	CONST robtarget Target_4220:=[[214.1,79.9,-54.2],[-0.0760679807605466,0.65526150182537,0.742837140883982,-0.114188478630225],[0,0,0,1],[9E+09,9E+09,9E+09,9E+09,9E+09,9E+09]];
	CONST robtarget Target_4230:=[[214.1,84.6,-54.5],[-0.0747816180925732,0.654610534044765,0.743306705241576,-0.115706094290646],[0,0,0,1],[9E+09,9E+09,9E+09,9E+09,9E+09,9E+09]];
	CONST robtarget Target_4240:=[[214.1,89.3,-54.9],[-0.073531882239943,0.653955613371436,0.743775907688082,-0.117185823276578],[0,0,0,1],[9E+09,9E+09,9E+09,9E+09,9E+09,9E+09]];
	CONST robtarget Target_4250:=[[214.1,94,-55.2],[-0.0722505034042859,0.653283696519975,0.744251094825556,-0.118703767716048],[0,0,0,1],[9E+09,9E+09,9E+09,9E+09,9E+09,9E+09]];
	CONST robtarget Target_4260:=[[214.1,98.7,-55.6],[-0.0709718230450671,0.652600969502751,0.744729273860509,-0.120221809971935],[0,0,0,1],[9E+09,9E+09,9E+09,9E+09,9E+09,9E+09]];
	CONST robtarget Target_4270:=[[214.1,103.4,-56.1],[-0.0697368456344226,0.651911675562493,0.745207121516542,-0.121713950175375],[0,0,0,1],[9E+09,9E+09,9E+09,9E+09,9E+09,9E+09]];
	CONST robtarget Target_4280:=[[214.1,108.1,-56.5],[-0.0684638092553564,0.65120670448846,0.745691861757032,-0.123232228580258],[0,0,0,1],[9E+09,9E+09,9E+09,9E+09,9E+09,9E+09]];
	CONST robtarget Target_4290:=[[214.1,112.9,-56.9],[-0.0672019671558274,0.650478513802981,0.746187667457493,-0.12476202797886],[0,0,0,1],[9E+09,9E+09,9E+09,9E+09,9E+09,9E+09]];
	CONST robtarget Target_4300:=[[214.1,117.6,-57.4],[-0.0659415982702471,0.649747743117887,0.746679097173527,-0.126292920525678],[0,0,0,1],[9E+09,9E+09,9E+09,9E+09,9E+09,9E+09]];
	CONST robtarget Target_4310:=[[214.1,122.3,-57.9],[-0.064724629163582,0.649009411435852,0.747171328797483,-0.127798715448665],[0,0,0,1],[9E+09,9E+09,9E+09,9E+09,9E+09,9E+09]];
	CONST robtarget Target_4320:=[[214.1,126.9,-58.4],[-0.0634688183068436,0.648264268897657,0.747662116568994,-0.129330994819074],[0,0,0,1],[9E+09,9E+09,9E+09,9E+09,9E+09,9E+09]];
	CONST robtarget Target_4330:=[[214.1,131.6,-59],[-0.0622181375236594,0.647496731507395,0.748165675952307,-0.13086255146968],[0,0,0,1],[9E+09,9E+09,9E+09,9E+09,9E+09,9E+09]];
	CONST robtarget Target_4340:=[[214.1,136.3,-59.5],[-0.0610108478057296,0.646720866963663,0.748670915845893,-0.132369393933289],[0,0,0,1],[9E+09,9E+09,9E+09,9E+09,9E+09,9E+09]];
	CONST robtarget Target_4350:=[[214.1,141,-60.1],[-0.0597731615365629,0.645924637221304,0.749183165378491,-0.133914588092245],[0,0,0,1],[9E+09,9E+09,9E+09,9E+09,9E+09,9E+09]];
	CONST robtarget Target_4360:=[[214.1,145.7,-60.7],[-0.0585391714057714,0.64511482893062,0.749700327915236,-0.135460109363351],[0,0,0,1],[9E+09,9E+09,9E+09,9E+09,9E+09,9E+09]];
	CONST robtarget Target_4370:=[[214.1,150.4,-61.3],[-0.0573428290888,0.644298492896021,0.750220650493769,-0.136967980114748],[0,0,0,1],[9E+09,9E+09,9E+09,9E+09,9E+09,9E+09]];
	CONST robtarget Target_4380:=[[214.1,155.2,-61.9],[-0.0561242209793799,0.643446414332673,0.750757651605653,-0.138527009126195],[0,0,0,1],[9E+09,9E+09,9E+09,9E+09,9E+09,9E+09]];
	CONST robtarget Target_4390:=[[214.1,159.9,-62.6],[-0.0549022874737579,0.642593676162974,0.751291241769304,-0.140073467245733],[0,0,0,1],[9E+09,9E+09,9E+09,9E+09,9E+09,9E+09]];
	CONST robtarget Target_4400:=[[214.1,164.6,-63.3],[-0.0536899475070816,0.641723004287069,0.751830248201575,-0.141634223246443],[0,0,0,1],[9E+09,9E+09,9E+09,9E+09,9E+09,9E+09]];
	CONST robtarget Target_4410:=[[214.1,169.3,-64],[-0.0525156005654393,0.640844533278809,0.752373783438205,-0.143157556066027],[0,0,0,1],[9E+09,9E+09,9E+09,9E+09,9E+09,9E+09]];
	CONST robtarget Target_4420:=[[214.1,174,-64.7],[-0.0513121794704837,0.639942656609551,0.752925495500269,-0.144719227178605],[0,0,0,1],[9E+09,9E+09,9E+09,9E+09,9E+09,9E+09]];
	CONST robtarget Target_4430:=[[214.1,178.7,-65.4],[-0.0501135494154515,0.639024535867129,0.753483945328914,-0.146281300432967],[0,0,0,1],[9E+09,9E+09,9E+09,9E+09,9E+09,9E+09]];
	CONST robtarget Target_4440:=[[214.1,183.4,-66.2],[-0.0489533985393246,0.638097583939901,0.754048044913025,-0.147805900099946],[0,0,0,1],[9E+09,9E+09,9E+09,9E+09,9E+09,9E+09]];
	CONST robtarget Target_4450:=[[214.1,188.1,-66.9],[-0.0477695461555189,0.63714240176872,0.754620547485047,-0.149383598972081],[0,0,0,1],[9E+09,9E+09,9E+09,9E+09,9E+09,9E+09]];
	CONST robtarget Target_4460:=[[214.1,192.8,-67.7],[-0.0465864465741739,0.636172890269665,0.755201164633342,-0.15094687018278],[0,0,0,1],[9E+09,9E+09,9E+09,9E+09,9E+09,9E+09]];
	CONST robtarget Target_4470:=[[214.1,197.5,-68.6],[-0.0454467284791908,0.635189863884349,0.755788257500963,-0.152487840540739],[0,0,0,1],[9E+09,9E+09,9E+09,9E+09,9E+09,9E+09]];
	CONST robtarget Target_4480:=[[214.1,202.2,-69.4],[-0.0442793548151249,0.634180120150372,0.756384963217846,-0.154067197550788],[0,0,0,1],[9E+09,9E+09,9E+09,9E+09,9E+09,9E+09]];
	CONST robtarget Target_4490:=[[214.1,206.9,-70.2],[-0.0431220973517324,0.633147478237495,0.756990026801105,-0.155662631498866],[0,0,0,1],[9E+09,9E+09,9E+09,9E+09,9E+09,9E+09]];
	CONST robtarget Target_4500:=[[214.1,211.6,-71.1],[-0.0419668302732848,0.632098525050186,0.757604653725667,-0.15724321428731],[0,0,0,1],[9E+09,9E+09,9E+09,9E+09,9E+09,9E+09]];
	CONST robtarget Target_4510:=[[214.1,216.3,-72],[-0.0408551063250609,0.631033669006859,0.758227646379614,-0.158802409089222],[0,0,0,1],[9E+09,9E+09,9E+09,9E+09,9E+09,9E+09]];
	CONST robtarget Target_4520:=[[214.1,221,-72.9],[-0.0397129990436774,0.629943181324887,0.758861906903818,-0.160384139675776],[0,0,0,1],[9E+09,9E+09,9E+09,9E+09,9E+09,9E+09]];
	CONST robtarget Target_4530:=[[214.1,225.7,-73.9],[-0.0385817057921211,0.628827052341548,0.759506197346856,-0.161982487983516],[0,0,0,1],[9E+09,9E+09,9E+09,9E+09,9E+09,9E+09]];
	CONST robtarget Target_4540:=[[214.1,230.4,-74.8],[-0.0374905350461494,0.627696847333574,0.760160850569989,-0.163543905084095],[0,0,0,1],[9E+09,9E+09,9E+09,9E+09,9E+09,9E+09]];
	CONST robtarget Target_4550:=[[214.1,235.1,-75.8],[-0.036377410933379,0.626530843722664,0.760827103763876,-0.165160237394547],[0,0,0,1],[9E+09,9E+09,9E+09,9E+09,9E+09,9E+09]];
	CONST robtarget Target_4560:=[[214.1,239.8,-76.8],[-0.0352685565372593,0.625344750184507,0.761505650251853,-0.166760957573877],[0,0,0,1],[9E+09,9E+09,9E+09,9E+09,9E+09,9E+09]];
	CONST robtarget Target_4570:=[[214.1,244.5,-77.8],[-0.0341712180146319,0.624129563242526,0.762196213319151,-0.168379180862828],[0,0,0,1],[9E+09,9E+09,9E+09,9E+09,9E+09,9E+09]];
	CONST robtarget Target_4580:=[[218.8,244.2,-79.1],[-0.0352789013652378,0.61925527973127,0.766168461703898,-0.168119558450798],[0,0,0,1],[9E+09,9E+09,9E+09,9E+09,9E+09,9E+09]];
	CONST robtarget Target_4590:=[[223.5,243.9,-80.3],[-0.0363420920703788,0.614382529573869,0.770085191873047,-0.167875420941287],[0,0,0,1],[9E+09,9E+09,9E+09,9E+09,9E+09,9E+09]];
	CONST robtarget Target_4600:=[[228.2,243.6,-81.6],[-0.0374001271246908,0.609513532222938,0.773944668193309,-0.167642879667832],[0,0,0,1],[9E+09,9E+09,9E+09,9E+09,9E+09,9E+09]];
	CONST robtarget Target_4610:=[[232.9,243.3,-82.8],[-0.0384493332726948,0.604654398226158,0.777746844476721,-0.167405356494801],[0,0,0,1],[9E+09,9E+09,9E+09,9E+09,9E+09,9E+09]];
	CONST robtarget Target_4620:=[[237.6,243,-84.1],[-0.0394894517675504,0.599806981726168,0.781491317968587,-0.167163057555683],[0,0,0,1],[9E+09,9E+09,9E+09,9E+09,9E+09,9E+09]];
	CONST robtarget Target_4630:=[[242.4,242.7,-85.3],[-0.0405424217596268,0.594868736122905,0.78525682561266,-0.166910804473919],[0,0,0,1],[9E+09,9E+09,9E+09,9E+09,9E+09,9E+09]];
	CONST robtarget Target_4640:=[[247.1,242.4,-86.6],[-0.0415634621821783,0.590050377687373,0.788883798273689,-0.166659482849602],[0,0,0,1],[9E+09,9E+09,9E+09,9E+09,9E+09,9E+09]];
	CONST robtarget Target_4650:=[[251.8,242.1,-87.8],[-0.0426055282136537,0.585257721214646,0.792452473450789,-0.166364798097438],[0,0,0,1],[9E+09,9E+09,9E+09,9E+09,9E+09,9E+09]];
	CONST robtarget Target_4660:=[[256.5,241.9,-89.1],[-0.0436128251589251,0.580445150786425,0.795984264824474,-0.166103577812228],[0,0,0,1],[9E+09,9E+09,9E+09,9E+09,9E+09,9E+09]];
	CONST robtarget Target_4670:=[[261.2,241.6,-90.3],[-0.044603962147879,0.575681451164459,0.799436294963406,-0.165840174991093],[0,0,0,1],[9E+09,9E+09,9E+09,9E+09,9E+09,9E+09]];
	CONST robtarget Target_4680:=[[265.9,241.2,-91.6],[-0.0455781193684878,0.570971841278474,0.802806750959846,-0.165575095093428],[0,0,0,1],[9E+09,9E+09,9E+09,9E+09,9E+09,9E+09]];
	CONST robtarget Target_4690:=[[270.7,241,-92.8],[-0.04657611167879,0.566118569710976,0.806236496288795,-0.165297135187669],[0,0,0,1],[9E+09,9E+09,9E+09,9E+09,9E+09,9E+09]];
	CONST robtarget Target_4700:=[[275.4,240.7,-94.1],[-0.0475652784406573,0.561433672938044,0.809512308110473,-0.164983630084364],[0,0,0,1],[9E+09,9E+09,9E+09,9E+09,9E+09,9E+09]];
	CONST robtarget Target_4710:=[[280.1,240.4,-95.3],[-0.0485138773113708,0.556766097158342,0.812729634716316,-0.164707187509133],[0,0,0,1],[9E+09,9E+09,9E+09,9E+09,9E+09,9E+09]];
	CONST robtarget Target_4720:=[[284.8,240.1,-96.6],[-0.0494516568369335,0.552125800136082,0.815889114350191,-0.164428061914728],[0,0,0,1],[9E+09,9E+09,9E+09,9E+09,9E+09,9E+09]];
	CONST robtarget Target_4730:=[[289.5,239.8,-97.8],[-0.0503785277368699,0.547513991237142,0.818991071679431,-0.164146452450295],[0,0,0,1],[9E+09,9E+09,9E+09,9E+09,9E+09,9E+09]];
	CONST robtarget Target_4740:=[[294.2,239.5,-99.1],[-0.0512944143707967,0.54293181630632,0.822035880563232,-0.163862555098194],[0,0,0,1],[9E+09,9E+09,9E+09,9E+09,9E+09,9E+09]];
	CONST robtarget Target_4750:=[[299,239.2,-100.3],[-0.0522188939240138,0.538281296648858,0.82508859631501,-0.163570293838167],[0,0,0,1],[9E+09,9E+09,9E+09,9E+09,9E+09,9E+09]];
	CONST robtarget Target_4760:=[[303.7,238.9,-101.6],[-0.0531406589164049,0.533770858467849,0.828019948764244,-0.16324124928732],[0,0,0,1],[9E+09,9E+09,9E+09,9E+09,9E+09,9E+09]];
    !***********************************************************
    !
    ! Module:  test
    !
    ! Description:
    !   <Insert description>
    !
    ! Author: ModuleWriter
    ! Version: 1.0
    !
    !***********************************************************


    !***********************************************************
    !
    ! Procedure main
    !
    !   This is the entry point of your program
    !
    !***********************************************************
    PROC main()
        Path_10;
      !Add your code here
    ENDPROC
      PROC Path_10()
SetDO drillDone,0;
MoveAbsJ jHome, v100, fine, tool0\WObj:= wobj0;
WaitTime 2;
confL \Off;
confJ \Off;
        MoveJ RelTool(Target_10,0,0,-10),v60,z10,DrillTool\WObj:=FakeWing;
SetDO drillDone,1;
WaitUntil drillDone = 0;
        MoveL Target_10,v30,fine,DrillTool\WObj:=FakeWing;
SetDO drillDone,1;
WaitUntil drillDone = 0;
        MoveL RelTool(Target_10,0,0,-10),v30,z10,DrillTool\WObj:=FakeWing;
        MoveL RelTool(Target_20,0,0,-10),v30,z10,DrillTool\WObj:=FakeWing;
        MoveL Target_20,v30,fine,DrillTool\WObj:=FakeWing;
SetDO drillDone,1;
WaitUntil drillDone = 0;
        MoveL RelTool(Target_20,0,0,-10),v30,z10,DrillTool\WObj:=FakeWing;
        MoveL RelTool(Target_30,0,0,-10),v30,z10,DrillTool\WObj:=FakeWing;
        MoveL Target_30,v30,fine,DrillTool\WObj:=FakeWing;
SetDO drillDone,1;
WaitUntil drillDone = 0;
        MoveL RelTool(Target_30,0,0,-10),v30,z10,DrillTool\WObj:=FakeWing;
        MoveL RelTool(Target_40,0,0,-10),v30,z10,DrillTool\WObj:=FakeWing;
        MoveL Target_40,v30,fine,DrillTool\WObj:=FakeWing;
SetDO drillDone,1;
WaitUntil drillDone = 0;
        MoveL RelTool(Target_40,0,0,-10),v30,z10,DrillTool\WObj:=FakeWing;
        MoveL RelTool(Target_50,0,0,-10),v30,z10,DrillTool\WObj:=FakeWing;
        MoveL Target_50,v30,fine,DrillTool\WObj:=FakeWing;
SetDO drillDone,1;
WaitUntil drillDone = 0;
        MoveL RelTool(Target_50,0,0,-10),v30,z10,DrillTool\WObj:=FakeWing;
        MoveL RelTool(Target_60,0,0,-10),v30,z10,DrillTool\WObj:=FakeWing;
        MoveL Target_60,v30,fine,DrillTool\WObj:=FakeWing;
SetDO drillDone,1;
WaitUntil drillDone = 0;
        MoveL RelTool(Target_60,0,0,-10),v30,z10,DrillTool\WObj:=FakeWing;
        MoveL RelTool(Target_70,0,0,-10),v30,z10,DrillTool\WObj:=FakeWing;
        MoveL Target_70,v30,fine,DrillTool\WObj:=FakeWing;
SetDO drillDone,1;
WaitUntil drillDone = 0;
        MoveL RelTool(Target_70,0,0,-10),v30,z10,DrillTool\WObj:=FakeWing;
        MoveL RelTool(Target_80,0,0,-10),v30,z10,DrillTool\WObj:=FakeWing;
        MoveL Target_80,v30,fine,DrillTool\WObj:=FakeWing;
SetDO drillDone,1;
WaitUntil drillDone = 0;
        MoveL RelTool(Target_80,0,0,-10),v30,z10,DrillTool\WObj:=FakeWing;
        MoveL RelTool(Target_90,0,0,-10),v30,z10,DrillTool\WObj:=FakeWing;
        MoveL Target_90,v30,fine,DrillTool\WObj:=FakeWing;
SetDO drillDone,1;
WaitUntil drillDone = 0;
        MoveL RelTool(Target_90,0,0,-10),v30,z10,DrillTool\WObj:=FakeWing;
        MoveL RelTool(Target_100,0,0,-10),v30,z10,DrillTool\WObj:=FakeWing;
        MoveL Target_100,v30,fine,DrillTool\WObj:=FakeWing;
SetDO drillDone,1;
WaitUntil drillDone = 0;
        MoveL RelTool(Target_100,0,0,-10),v30,z10,DrillTool\WObj:=FakeWing;
        MoveL RelTool(Target_110,0,0,-10),v30,z10,DrillTool\WObj:=FakeWing;
        MoveL Target_110,v30,fine,DrillTool\WObj:=FakeWing;
SetDO drillDone,1;
WaitUntil drillDone = 0;
        MoveL RelTool(Target_110,0,0,-10),v30,z10,DrillTool\WObj:=FakeWing;
        MoveL RelTool(Target_120,0,0,-10),v30,z10,DrillTool\WObj:=FakeWing;
        MoveL Target_120,v30,fine,DrillTool\WObj:=FakeWing;
SetDO drillDone,1;
WaitUntil drillDone = 0;
        MoveL RelTool(Target_120,0,0,-10),v30,z10,DrillTool\WObj:=FakeWing;
        MoveL RelTool(Target_130,0,0,-10),v30,z10,DrillTool\WObj:=FakeWing;
        MoveL Target_130,v30,fine,DrillTool\WObj:=FakeWing;
SetDO drillDone,1;
WaitUntil drillDone = 0;
        MoveL RelTool(Target_130,0,0,-10),v30,z10,DrillTool\WObj:=FakeWing;
        MoveL RelTool(Target_140,0,0,-10),v30,z10,DrillTool\WObj:=FakeWing;
        MoveL Target_140,v30,fine,DrillTool\WObj:=FakeWing;
SetDO drillDone,1;
WaitUntil drillDone = 0;
        MoveL RelTool(Target_140,0,0,-10),v30,z10,DrillTool\WObj:=FakeWing;
        MoveL RelTool(Target_150,0,0,-10),v30,z10,DrillTool\WObj:=FakeWing;
        MoveL Target_150,v30,fine,DrillTool\WObj:=FakeWing;
SetDO drillDone,1;
WaitUntil drillDone = 0;
        MoveL RelTool(Target_150,0,0,-10),v30,z10,DrillTool\WObj:=FakeWing;
        MoveL RelTool(Target_160,0,0,-10),v30,z10,DrillTool\WObj:=FakeWing;
        MoveL Target_160,v30,fine,DrillTool\WObj:=FakeWing;
SetDO drillDone,1;
WaitUntil drillDone = 0;
        MoveL RelTool(Target_160,0,0,-10),v30,z10,DrillTool\WObj:=FakeWing;
        MoveL RelTool(Target_170,0,0,-10),v30,z10,DrillTool\WObj:=FakeWing;
        MoveL Target_170,v30,fine,DrillTool\WObj:=FakeWing;
SetDO drillDone,1;
WaitUntil drillDone = 0;
        MoveL RelTool(Target_170,0,0,-10),v30,z10,DrillTool\WObj:=FakeWing;
        MoveL RelTool(Target_180,0,0,-10),v30,z10,DrillTool\WObj:=FakeWing;
        MoveL Target_180,v30,fine,DrillTool\WObj:=FakeWing;
SetDO drillDone,1;
WaitUntil drillDone = 0;
        MoveL RelTool(Target_180,0,0,-10),v30,z10,DrillTool\WObj:=FakeWing;
        MoveL RelTool(Target_190,0,0,-10),v30,z10,DrillTool\WObj:=FakeWing;
        MoveL Target_190,v30,fine,DrillTool\WObj:=FakeWing;
SetDO drillDone,1;
WaitUntil drillDone = 0;
        MoveL RelTool(Target_190,0,0,-10),v30,z10,DrillTool\WObj:=FakeWing;
        MoveL RelTool(Target_200,0,0,-10),v30,z10,DrillTool\WObj:=FakeWing;
        MoveL Target_200,v30,fine,DrillTool\WObj:=FakeWing;
SetDO drillDone,1;
WaitUntil drillDone = 0;
        MoveL RelTool(Target_200,0,0,-10),v30,z10,DrillTool\WObj:=FakeWing;
        MoveL RelTool(Target_210,0,0,-10),v30,z10,DrillTool\WObj:=FakeWing;
        MoveL Target_210,v30,fine,DrillTool\WObj:=FakeWing;
SetDO drillDone,1;
WaitUntil drillDone = 0;
        MoveL RelTool(Target_210,0,0,-10),v30,z10,DrillTool\WObj:=FakeWing;
        MoveL RelTool(Target_220,0,0,-10),v30,z10,DrillTool\WObj:=FakeWing;
        MoveL Target_220,v30,fine,DrillTool\WObj:=FakeWing;
SetDO drillDone,1;
WaitUntil drillDone = 0;
        MoveL RelTool(Target_220,0,0,-10),v30,z10,DrillTool\WObj:=FakeWing;
        MoveL RelTool(Target_230,0,0,-10),v30,z10,DrillTool\WObj:=FakeWing;
        MoveL Target_230,v30,fine,DrillTool\WObj:=FakeWing;
SetDO drillDone,1;
WaitUntil drillDone = 0;
        MoveL RelTool(Target_230,0,0,-10),v30,z10,DrillTool\WObj:=FakeWing;
        MoveL RelTool(Target_240,0,0,-10),v30,z10,DrillTool\WObj:=FakeWing;
        MoveL Target_240,v30,fine,DrillTool\WObj:=FakeWing;
SetDO drillDone,1;
WaitUntil drillDone = 0;
        MoveL RelTool(Target_240,0,0,-10),v30,z10,DrillTool\WObj:=FakeWing;
        MoveL RelTool(Target_250,0,0,-10),v30,z10,DrillTool\WObj:=FakeWing;
        MoveL Target_250,v30,fine,DrillTool\WObj:=FakeWing;
SetDO drillDone,1;
WaitUntil drillDone = 0;
        MoveL RelTool(Target_250,0,0,-10),v30,z10,DrillTool\WObj:=FakeWing;
        MoveL RelTool(Target_260,0,0,-10),v30,z10,DrillTool\WObj:=FakeWing;
        MoveL Target_260,v30,fine,DrillTool\WObj:=FakeWing;
SetDO drillDone,1;
WaitUntil drillDone = 0;
        MoveL RelTool(Target_260,0,0,-10),v30,z10,DrillTool\WObj:=FakeWing;
        MoveL RelTool(Target_270,0,0,-10),v30,z10,DrillTool\WObj:=FakeWing;
        MoveL Target_270,v30,fine,DrillTool\WObj:=FakeWing;
SetDO drillDone,1;
WaitUntil drillDone = 0;
        MoveL RelTool(Target_270,0,0,-10),v30,z10,DrillTool\WObj:=FakeWing;
        MoveL RelTool(Target_280,0,0,-10),v30,z10,DrillTool\WObj:=FakeWing;
        MoveL Target_280,v30,fine,DrillTool\WObj:=FakeWing;
SetDO drillDone,1;
WaitUntil drillDone = 0;
        MoveL RelTool(Target_280,0,0,-10),v30,z10,DrillTool\WObj:=FakeWing;
        MoveL RelTool(Target_290,0,0,-10),v30,z10,DrillTool\WObj:=FakeWing;
        MoveL Target_290,v30,fine,DrillTool\WObj:=FakeWing;
SetDO drillDone,1;
WaitUntil drillDone = 0;
        MoveL RelTool(Target_290,0,0,-10),v30,z10,DrillTool\WObj:=FakeWing;
        MoveL RelTool(Target_300,0,0,-10),v30,z10,DrillTool\WObj:=FakeWing;
        MoveL Target_300,v30,fine,DrillTool\WObj:=FakeWing;
SetDO drillDone,1;
WaitUntil drillDone = 0;
        MoveL RelTool(Target_300,0,0,-10),v30,z10,DrillTool\WObj:=FakeWing;
        MoveL RelTool(Target_310,0,0,-10),v30,z10,DrillTool\WObj:=FakeWing;
        MoveL Target_310,v30,fine,DrillTool\WObj:=FakeWing;
SetDO drillDone,1;
WaitUntil drillDone = 0;
        MoveL RelTool(Target_310,0,0,-10),v30,z10,DrillTool\WObj:=FakeWing;
        MoveL RelTool(Target_320,0,0,-10),v30,z10,DrillTool\WObj:=FakeWing;
        MoveL Target_320,v30,fine,DrillTool\WObj:=FakeWing;
SetDO drillDone,1;
WaitUntil drillDone = 0;
        MoveL RelTool(Target_320,0,0,-10),v30,z10,DrillTool\WObj:=FakeWing;
        MoveL RelTool(Target_330,0,0,-10),v30,z10,DrillTool\WObj:=FakeWing;
        MoveL Target_330,v30,fine,DrillTool\WObj:=FakeWing;
SetDO drillDone,1;
WaitUntil drillDone = 0;
        MoveL RelTool(Target_330,0,0,-10),v30,z10,DrillTool\WObj:=FakeWing;
        MoveL RelTool(Target_340,0,0,-10),v30,z10,DrillTool\WObj:=FakeWing;
        MoveL Target_340,v30,fine,DrillTool\WObj:=FakeWing;
SetDO drillDone,1;
WaitUntil drillDone = 0;
        MoveL RelTool(Target_340,0,0,-10),v30,z10,DrillTool\WObj:=FakeWing;
        MoveL RelTool(Target_350,0,0,-10),v30,z10,DrillTool\WObj:=FakeWing;
        MoveL Target_350,v30,fine,DrillTool\WObj:=FakeWing;
SetDO drillDone,1;
WaitUntil drillDone = 0;
        MoveL RelTool(Target_350,0,0,-10),v30,z10,DrillTool\WObj:=FakeWing;
        MoveL RelTool(Target_360,0,0,-10),v30,z10,DrillTool\WObj:=FakeWing;
        MoveL Target_360,v30,fine,DrillTool\WObj:=FakeWing;
SetDO drillDone,1;
WaitUntil drillDone = 0;
        MoveL RelTool(Target_360,0,0,-10),v30,z10,DrillTool\WObj:=FakeWing;
        MoveL RelTool(Target_370,0,0,-10),v30,z10,DrillTool\WObj:=FakeWing;
        MoveL Target_370,v30,fine,DrillTool\WObj:=FakeWing;
SetDO drillDone,1;
WaitUntil drillDone = 0;
        MoveL RelTool(Target_370,0,0,-10),v30,z10,DrillTool\WObj:=FakeWing;
        MoveL RelTool(Target_380,0,0,-10),v30,z10,DrillTool\WObj:=FakeWing;
        MoveL Target_380,v30,fine,DrillTool\WObj:=FakeWing;
SetDO drillDone,1;
WaitUntil drillDone = 0;
        MoveL RelTool(Target_380,0,0,-10),v30,z10,DrillTool\WObj:=FakeWing;
        MoveL RelTool(Target_390,0,0,-10),v30,z10,DrillTool\WObj:=FakeWing;
        MoveL Target_390,v30,fine,DrillTool\WObj:=FakeWing;
SetDO drillDone,1;
WaitUntil drillDone = 0;
        MoveL RelTool(Target_390,0,0,-10),v30,z10,DrillTool\WObj:=FakeWing;
        MoveL RelTool(Target_400,0,0,-10),v30,z10,DrillTool\WObj:=FakeWing;
        MoveL Target_400,v30,fine,DrillTool\WObj:=FakeWing;
SetDO drillDone,1;
WaitUntil drillDone = 0;
        MoveL RelTool(Target_400,0,0,-10),v30,z10,DrillTool\WObj:=FakeWing;
        MoveL RelTool(Target_410,0,0,-10),v30,z10,DrillTool\WObj:=FakeWing;
        MoveL Target_410,v30,fine,DrillTool\WObj:=FakeWing;
SetDO drillDone,1;
WaitUntil drillDone = 0;
        MoveL RelTool(Target_410,0,0,-10),v30,z10,DrillTool\WObj:=FakeWing;
        MoveL RelTool(Target_420,0,0,-10),v30,z10,DrillTool\WObj:=FakeWing;
        MoveL Target_420,v30,fine,DrillTool\WObj:=FakeWing;
SetDO drillDone,1;
WaitUntil drillDone = 0;
        MoveL RelTool(Target_420,0,0,-10),v30,z10,DrillTool\WObj:=FakeWing;
        MoveL RelTool(Target_430,0,0,-10),v30,z10,DrillTool\WObj:=FakeWing;
        MoveL Target_430,v30,fine,DrillTool\WObj:=FakeWing;
SetDO drillDone,1;
WaitUntil drillDone = 0;
        MoveL RelTool(Target_430,0,0,-10),v30,z10,DrillTool\WObj:=FakeWing;
        MoveL RelTool(Target_440,0,0,-10),v30,z10,DrillTool\WObj:=FakeWing;
        MoveL Target_440,v30,fine,DrillTool\WObj:=FakeWing;
SetDO drillDone,1;
WaitUntil drillDone = 0;
        MoveL RelTool(Target_440,0,0,-10),v30,z10,DrillTool\WObj:=FakeWing;
        MoveL RelTool(Target_450,0,0,-10),v30,z10,DrillTool\WObj:=FakeWing;
        MoveL Target_450,v30,fine,DrillTool\WObj:=FakeWing;
SetDO drillDone,1;
WaitUntil drillDone = 0;
        MoveL RelTool(Target_450,0,0,-10),v30,z10,DrillTool\WObj:=FakeWing;
        MoveL RelTool(Target_460,0,0,-10),v30,z10,DrillTool\WObj:=FakeWing;
        MoveL Target_460,v30,fine,DrillTool\WObj:=FakeWing;
SetDO drillDone,1;
WaitUntil drillDone = 0;
        MoveL RelTool(Target_460,0,0,-10),v30,z10,DrillTool\WObj:=FakeWing;
        MoveL RelTool(Target_470,0,0,-10),v30,z10,DrillTool\WObj:=FakeWing;
        MoveL Target_470,v30,fine,DrillTool\WObj:=FakeWing;
SetDO drillDone,1;
WaitUntil drillDone = 0;
        MoveL RelTool(Target_470,0,0,-10),v30,z10,DrillTool\WObj:=FakeWing;
        MoveL RelTool(Target_480,0,0,-10),v30,z10,DrillTool\WObj:=FakeWing;
        MoveL Target_480,v30,fine,DrillTool\WObj:=FakeWing;
SetDO drillDone,1;
WaitUntil drillDone = 0;
        MoveL RelTool(Target_480,0,0,-10),v30,z10,DrillTool\WObj:=FakeWing;
        MoveL RelTool(Target_490,0,0,-10),v30,z10,DrillTool\WObj:=FakeWing;
        MoveL Target_490,v30,fine,DrillTool\WObj:=FakeWing;
SetDO drillDone,1;
WaitUntil drillDone = 0;
        MoveL RelTool(Target_490,0,0,-10),v30,z10,DrillTool\WObj:=FakeWing;
        MoveL RelTool(Target_500,0,0,-10),v30,z10,DrillTool\WObj:=FakeWing;
        MoveL Target_500,v30,fine,DrillTool\WObj:=FakeWing;
SetDO drillDone,1;
WaitUntil drillDone = 0;
        MoveL RelTool(Target_500,0,0,-10),v30,z10,DrillTool\WObj:=FakeWing;
        MoveL RelTool(Target_510,0,0,-10),v30,z10,DrillTool\WObj:=FakeWing;
        MoveL Target_510,v30,fine,DrillTool\WObj:=FakeWing;
SetDO drillDone,1;
WaitUntil drillDone = 0;
        MoveL RelTool(Target_510,0,0,-10),v30,z10,DrillTool\WObj:=FakeWing;
        MoveL RelTool(Target_520,0,0,-10),v30,z10,DrillTool\WObj:=FakeWing;
        MoveL Target_520,v30,fine,DrillTool\WObj:=FakeWing;
SetDO drillDone,1;
WaitUntil drillDone = 0;
        MoveL RelTool(Target_520,0,0,-10),v30,z10,DrillTool\WObj:=FakeWing;
        MoveL RelTool(Target_530,0,0,-10),v30,z10,DrillTool\WObj:=FakeWing;
        MoveL Target_530,v30,fine,DrillTool\WObj:=FakeWing;
SetDO drillDone,1;
WaitUntil drillDone = 0;
        MoveL RelTool(Target_530,0,0,-10),v30,z10,DrillTool\WObj:=FakeWing;
        MoveL RelTool(Target_540,0,0,-10),v30,z10,DrillTool\WObj:=FakeWing;
        MoveL Target_540,v30,fine,DrillTool\WObj:=FakeWing;
SetDO drillDone,1;
WaitUntil drillDone = 0;
        MoveL RelTool(Target_540,0,0,-10),v30,z10,DrillTool\WObj:=FakeWing;
        MoveL RelTool(Target_550,0,0,-10),v30,z10,DrillTool\WObj:=FakeWing;
        MoveL Target_550,v30,fine,DrillTool\WObj:=FakeWing;
SetDO drillDone,1;
WaitUntil drillDone = 0;
        MoveL RelTool(Target_550,0,0,-10),v30,z10,DrillTool\WObj:=FakeWing;
        MoveL RelTool(Target_560,0,0,-10),v30,z10,DrillTool\WObj:=FakeWing;
        MoveL Target_560,v30,fine,DrillTool\WObj:=FakeWing;
SetDO drillDone,1;
WaitUntil drillDone = 0;
        MoveL RelTool(Target_560,0,0,-10),v30,z10,DrillTool\WObj:=FakeWing;
        MoveL RelTool(Target_570,0,0,-10),v30,z10,DrillTool\WObj:=FakeWing;
        MoveL Target_570,v30,fine,DrillTool\WObj:=FakeWing;
SetDO drillDone,1;
WaitUntil drillDone = 0;
        MoveL RelTool(Target_570,0,0,-10),v30,z10,DrillTool\WObj:=FakeWing;
        MoveL RelTool(Target_580,0,0,-10),v30,z10,DrillTool\WObj:=FakeWing;
        MoveL Target_580,v30,fine,DrillTool\WObj:=FakeWing;
SetDO drillDone,1;
WaitUntil drillDone = 0;
        MoveL RelTool(Target_580,0,0,-10),v30,z10,DrillTool\WObj:=FakeWing;
        MoveL RelTool(Target_590,0,0,-10),v30,z10,DrillTool\WObj:=FakeWing;
        MoveL Target_590,v30,fine,DrillTool\WObj:=FakeWing;
SetDO drillDone,1;
WaitUntil drillDone = 0;
        MoveL RelTool(Target_590,0,0,-10),v30,z10,DrillTool\WObj:=FakeWing;
        MoveL RelTool(Target_600,0,0,-10),v30,z10,DrillTool\WObj:=FakeWing;
        MoveL Target_600,v30,fine,DrillTool\WObj:=FakeWing;
SetDO drillDone,1;
WaitUntil drillDone = 0;
        MoveL RelTool(Target_600,0,0,-10),v30,z10,DrillTool\WObj:=FakeWing;
        MoveL RelTool(Target_610,0,0,-10),v30,z10,DrillTool\WObj:=FakeWing;
        MoveL Target_610,v30,fine,DrillTool\WObj:=FakeWing;
SetDO drillDone,1;
WaitUntil drillDone = 0;
        MoveL RelTool(Target_610,0,0,-10),v30,z10,DrillTool\WObj:=FakeWing;
        MoveL RelTool(Target_620,0,0,-10),v30,z10,DrillTool\WObj:=FakeWing;
        MoveL Target_620,v30,fine,DrillTool\WObj:=FakeWing;
SetDO drillDone,1;
WaitUntil drillDone = 0;
        MoveL RelTool(Target_620,0,0,-10),v30,z10,DrillTool\WObj:=FakeWing;
        MoveL RelTool(Target_630,0,0,-10),v30,z10,DrillTool\WObj:=FakeWing;
        MoveL Target_630,v30,fine,DrillTool\WObj:=FakeWing;
SetDO drillDone,1;
WaitUntil drillDone = 0;
        MoveL RelTool(Target_630,0,0,-10),v30,z10,DrillTool\WObj:=FakeWing;
        MoveL RelTool(Target_640,0,0,-10),v30,z10,DrillTool\WObj:=FakeWing;
        MoveL Target_640,v30,fine,DrillTool\WObj:=FakeWing;
SetDO drillDone,1;
WaitUntil drillDone = 0;
        MoveL RelTool(Target_640,0,0,-10),v30,z10,DrillTool\WObj:=FakeWing;
        MoveL RelTool(Target_650,0,0,-10),v30,z10,DrillTool\WObj:=FakeWing;
        MoveL Target_650,v30,fine,DrillTool\WObj:=FakeWing;
SetDO drillDone,1;
WaitUntil drillDone = 0;
        MoveL RelTool(Target_650,0,0,-10),v30,z10,DrillTool\WObj:=FakeWing;
        MoveL RelTool(Target_660,0,0,-10),v30,z10,DrillTool\WObj:=FakeWing;
        MoveL Target_660,v30,fine,DrillTool\WObj:=FakeWing;
SetDO drillDone,1;
WaitUntil drillDone = 0;
        MoveL RelTool(Target_660,0,0,-10),v30,z10,DrillTool\WObj:=FakeWing;
        MoveL RelTool(Target_670,0,0,-10),v30,z10,DrillTool\WObj:=FakeWing;
        MoveL Target_670,v30,fine,DrillTool\WObj:=FakeWing;
SetDO drillDone,1;
WaitUntil drillDone = 0;
        MoveL RelTool(Target_670,0,0,-10),v30,z10,DrillTool\WObj:=FakeWing;
        MoveL RelTool(Target_680,0,0,-10),v30,z10,DrillTool\WObj:=FakeWing;
        MoveL Target_680,v30,fine,DrillTool\WObj:=FakeWing;
SetDO drillDone,1;
WaitUntil drillDone = 0;
        MoveL RelTool(Target_680,0,0,-10),v30,z10,DrillTool\WObj:=FakeWing;
        MoveL RelTool(Target_690,0,0,-10),v30,z10,DrillTool\WObj:=FakeWing;
        MoveL Target_690,v30,fine,DrillTool\WObj:=FakeWing;
SetDO drillDone,1;
WaitUntil drillDone = 0;
        MoveL RelTool(Target_690,0,0,-10),v30,z10,DrillTool\WObj:=FakeWing;
        MoveL RelTool(Target_700,0,0,-10),v30,z10,DrillTool\WObj:=FakeWing;
        MoveL Target_700,v30,fine,DrillTool\WObj:=FakeWing;
SetDO drillDone,1;
WaitUntil drillDone = 0;
        MoveL RelTool(Target_700,0,0,-10),v30,z10,DrillTool\WObj:=FakeWing;
        MoveL RelTool(Target_710,0,0,-10),v30,z10,DrillTool\WObj:=FakeWing;
        MoveL Target_710,v30,fine,DrillTool\WObj:=FakeWing;
SetDO drillDone,1;
WaitUntil drillDone = 0;
        MoveL RelTool(Target_710,0,0,-10),v30,z10,DrillTool\WObj:=FakeWing;
        MoveL RelTool(Target_720,0,0,-10),v30,z10,DrillTool\WObj:=FakeWing;
        MoveL Target_720,v30,fine,DrillTool\WObj:=FakeWing;
SetDO drillDone,1;
WaitUntil drillDone = 0;
        MoveL RelTool(Target_720,0,0,-10),v30,z10,DrillTool\WObj:=FakeWing;
        MoveL RelTool(Target_730,0,0,-10),v30,z10,DrillTool\WObj:=FakeWing;
        MoveL Target_730,v30,fine,DrillTool\WObj:=FakeWing;
SetDO drillDone,1;
WaitUntil drillDone = 0;
        MoveL RelTool(Target_730,0,0,-10),v30,z10,DrillTool\WObj:=FakeWing;
        MoveL RelTool(Target_740,0,0,-10),v30,z10,DrillTool\WObj:=FakeWing;
        MoveL Target_740,v30,fine,DrillTool\WObj:=FakeWing;
SetDO drillDone,1;
WaitUntil drillDone = 0;
        MoveL RelTool(Target_740,0,0,-10),v30,z10,DrillTool\WObj:=FakeWing;
        MoveL RelTool(Target_750,0,0,-10),v30,z10,DrillTool\WObj:=FakeWing;
        MoveL Target_750,v30,fine,DrillTool\WObj:=FakeWing;
SetDO drillDone,1;
WaitUntil drillDone = 0;
        MoveL RelTool(Target_750,0,0,-10),v30,z10,DrillTool\WObj:=FakeWing;
        MoveL RelTool(Target_760,0,0,-10),v30,z10,DrillTool\WObj:=FakeWing;
        MoveL Target_760,v30,fine,DrillTool\WObj:=FakeWing;
SetDO drillDone,1;
WaitUntil drillDone = 0;
        MoveL RelTool(Target_760,0,0,-10),v30,z10,DrillTool\WObj:=FakeWing;
        MoveL RelTool(Target_770,0,0,-10),v30,z10,DrillTool\WObj:=FakeWing;
        MoveL Target_770,v30,fine,DrillTool\WObj:=FakeWing;
SetDO drillDone,1;
WaitUntil drillDone = 0;
        MoveL RelTool(Target_770,0,0,-10),v30,z10,DrillTool\WObj:=FakeWing;
        MoveL RelTool(Target_780,0,0,-10),v30,z10,DrillTool\WObj:=FakeWing;
        MoveL Target_780,v30,fine,DrillTool\WObj:=FakeWing;
SetDO drillDone,1;
WaitUntil drillDone = 0;
        MoveL RelTool(Target_780,0,0,-10),v30,z10,DrillTool\WObj:=FakeWing;
        MoveL RelTool(Target_790,0,0,-10),v30,z10,DrillTool\WObj:=FakeWing;
        MoveL Target_790,v30,fine,DrillTool\WObj:=FakeWing;
SetDO drillDone,1;
WaitUntil drillDone = 0;
        MoveL RelTool(Target_790,0,0,-10),v30,z10,DrillTool\WObj:=FakeWing;
        MoveL RelTool(Target_800,0,0,-10),v30,z10,DrillTool\WObj:=FakeWing;
        MoveL Target_800,v30,fine,DrillTool\WObj:=FakeWing;
SetDO drillDone,1;
WaitUntil drillDone = 0;
        MoveL RelTool(Target_800,0,0,-10),v30,z10,DrillTool\WObj:=FakeWing;
        MoveL RelTool(Target_810,0,0,-10),v30,z10,DrillTool\WObj:=FakeWing;
        MoveL Target_810,v30,fine,DrillTool\WObj:=FakeWing;
SetDO drillDone,1;
WaitUntil drillDone = 0;
        MoveL RelTool(Target_810,0,0,-10),v30,z10,DrillTool\WObj:=FakeWing;
        MoveL RelTool(Target_820,0,0,-10),v30,z10,DrillTool\WObj:=FakeWing;
        MoveL Target_820,v30,fine,DrillTool\WObj:=FakeWing;
SetDO drillDone,1;
WaitUntil drillDone = 0;
        MoveL RelTool(Target_820,0,0,-10),v30,z10,DrillTool\WObj:=FakeWing;
        MoveL RelTool(Target_830,0,0,-10),v30,z10,DrillTool\WObj:=FakeWing;
        MoveL Target_830,v30,fine,DrillTool\WObj:=FakeWing;
SetDO drillDone,1;
WaitUntil drillDone = 0;
        MoveL RelTool(Target_830,0,0,-10),v30,z10,DrillTool\WObj:=FakeWing;
        MoveL RelTool(Target_840,0,0,-10),v30,z10,DrillTool\WObj:=FakeWing;
        MoveL Target_840,v30,fine,DrillTool\WObj:=FakeWing;
SetDO drillDone,1;
WaitUntil drillDone = 0;
        MoveL RelTool(Target_840,0,0,-10),v30,z10,DrillTool\WObj:=FakeWing;
        MoveL RelTool(Target_850,0,0,-10),v30,z10,DrillTool\WObj:=FakeWing;
        MoveL Target_850,v30,fine,DrillTool\WObj:=FakeWing;
SetDO drillDone,1;
WaitUntil drillDone = 0;
        MoveL RelTool(Target_850,0,0,-10),v30,z10,DrillTool\WObj:=FakeWing;
        MoveL RelTool(Target_860,0,0,-10),v30,z10,DrillTool\WObj:=FakeWing;
        MoveL Target_860,v30,fine,DrillTool\WObj:=FakeWing;
SetDO drillDone,1;
WaitUntil drillDone = 0;
        MoveL RelTool(Target_860,0,0,-10),v30,z10,DrillTool\WObj:=FakeWing;
        MoveL RelTool(Target_870,0,0,-10),v30,z10,DrillTool\WObj:=FakeWing;
        MoveL Target_870,v30,fine,DrillTool\WObj:=FakeWing;
SetDO drillDone,1;
WaitUntil drillDone = 0;
        MoveL RelTool(Target_870,0,0,-10),v30,z10,DrillTool\WObj:=FakeWing;
        MoveL RelTool(Target_880,0,0,-10),v30,z10,DrillTool\WObj:=FakeWing;
        MoveL Target_880,v30,fine,DrillTool\WObj:=FakeWing;
SetDO drillDone,1;
WaitUntil drillDone = 0;
        MoveL RelTool(Target_880,0,0,-10),v30,z10,DrillTool\WObj:=FakeWing;
        MoveL RelTool(Target_890,0,0,-10),v30,z10,DrillTool\WObj:=FakeWing;
        MoveL Target_890,v30,fine,DrillTool\WObj:=FakeWing;
SetDO drillDone,1;
WaitUntil drillDone = 0;
        MoveL RelTool(Target_890,0,0,-10),v30,z10,DrillTool\WObj:=FakeWing;
        MoveL RelTool(Target_900,0,0,-10),v30,z10,DrillTool\WObj:=FakeWing;
        MoveL Target_900,v30,fine,DrillTool\WObj:=FakeWing;
SetDO drillDone,1;
WaitUntil drillDone = 0;
        MoveL RelTool(Target_900,0,0,-10),v30,z10,DrillTool\WObj:=FakeWing;
        MoveL RelTool(Target_910,0,0,-10),v30,z10,DrillTool\WObj:=FakeWing;
        MoveL Target_910,v30,fine,DrillTool\WObj:=FakeWing;
SetDO drillDone,1;
WaitUntil drillDone = 0;
        MoveL RelTool(Target_910,0,0,-10),v30,z10,DrillTool\WObj:=FakeWing;
        MoveL RelTool(Target_920,0,0,-10),v30,z10,DrillTool\WObj:=FakeWing;
        MoveL Target_920,v30,fine,DrillTool\WObj:=FakeWing;
SetDO drillDone,1;
WaitUntil drillDone = 0;
        MoveL RelTool(Target_920,0,0,-10),v30,z10,DrillTool\WObj:=FakeWing;
        MoveL RelTool(Target_930,0,0,-10),v30,z10,DrillTool\WObj:=FakeWing;
        MoveL Target_930,v30,fine,DrillTool\WObj:=FakeWing;
SetDO drillDone,1;
WaitUntil drillDone = 0;
        MoveL RelTool(Target_930,0,0,-10),v30,z10,DrillTool\WObj:=FakeWing;
        MoveL RelTool(Target_940,0,0,-10),v30,z10,DrillTool\WObj:=FakeWing;
        MoveL Target_940,v30,fine,DrillTool\WObj:=FakeWing;
SetDO drillDone,1;
WaitUntil drillDone = 0;
        MoveL RelTool(Target_940,0,0,-10),v30,z10,DrillTool\WObj:=FakeWing;
        MoveL RelTool(Target_950,0,0,-10),v30,z10,DrillTool\WObj:=FakeWing;
        MoveL Target_950,v30,fine,DrillTool\WObj:=FakeWing;
SetDO drillDone,1;
WaitUntil drillDone = 0;
        MoveL RelTool(Target_950,0,0,-10),v30,z10,DrillTool\WObj:=FakeWing;
        MoveL RelTool(Target_960,0,0,-10),v30,z10,DrillTool\WObj:=FakeWing;
        MoveL Target_960,v30,fine,DrillTool\WObj:=FakeWing;
SetDO drillDone,1;
WaitUntil drillDone = 0;
        MoveL RelTool(Target_960,0,0,-10),v30,z10,DrillTool\WObj:=FakeWing;
        MoveL RelTool(Target_970,0,0,-10),v30,z10,DrillTool\WObj:=FakeWing;
        MoveL Target_970,v30,fine,DrillTool\WObj:=FakeWing;
SetDO drillDone,1;
WaitUntil drillDone = 0;
        MoveL RelTool(Target_970,0,0,-10),v30,z10,DrillTool\WObj:=FakeWing;
        MoveL RelTool(Target_980,0,0,-10),v30,z10,DrillTool\WObj:=FakeWing;
        MoveL Target_980,v30,fine,DrillTool\WObj:=FakeWing;
SetDO drillDone,1;
WaitUntil drillDone = 0;
        MoveL RelTool(Target_980,0,0,-10),v30,z10,DrillTool\WObj:=FakeWing;
        MoveL RelTool(Target_990,0,0,-10),v30,z10,DrillTool\WObj:=FakeWing;
        MoveL Target_990,v30,fine,DrillTool\WObj:=FakeWing;
SetDO drillDone,1;
WaitUntil drillDone = 0;
        MoveL RelTool(Target_990,0,0,-10),v30,z10,DrillTool\WObj:=FakeWing;
        MoveL RelTool(Target_1000,0,0,-10),v30,z10,DrillTool\WObj:=FakeWing;
        MoveL Target_1000,v30,fine,DrillTool\WObj:=FakeWing;
SetDO drillDone,1;
WaitUntil drillDone = 0;
        MoveL RelTool(Target_1000,0,0,-10),v30,z10,DrillTool\WObj:=FakeWing;
        MoveL RelTool(Target_1010,0,0,-10),v30,z10,DrillTool\WObj:=FakeWing;
        MoveL Target_1010,v30,fine,DrillTool\WObj:=FakeWing;
SetDO drillDone,1;
WaitUntil drillDone = 0;
        MoveL RelTool(Target_1010,0,0,-10),v30,z10,DrillTool\WObj:=FakeWing;
        MoveL RelTool(Target_1020,0,0,-10),v30,z10,DrillTool\WObj:=FakeWing;
        MoveL Target_1020,v30,fine,DrillTool\WObj:=FakeWing;
SetDO drillDone,1;
WaitUntil drillDone = 0;
        MoveL RelTool(Target_1020,0,0,-10),v30,z10,DrillTool\WObj:=FakeWing;
        MoveL RelTool(Target_1030,0,0,-10),v30,z10,DrillTool\WObj:=FakeWing;
        MoveL Target_1030,v30,fine,DrillTool\WObj:=FakeWing;
SetDO drillDone,1;
WaitUntil drillDone = 0;
        MoveL RelTool(Target_1030,0,0,-10),v30,z10,DrillTool\WObj:=FakeWing;
        MoveL RelTool(Target_1040,0,0,-10),v30,z10,DrillTool\WObj:=FakeWing;
        MoveL Target_1040,v30,fine,DrillTool\WObj:=FakeWing;
SetDO drillDone,1;
WaitUntil drillDone = 0;
        MoveL RelTool(Target_1040,0,0,-10),v30,z10,DrillTool\WObj:=FakeWing;
        MoveL RelTool(Target_1050,0,0,-10),v30,z10,DrillTool\WObj:=FakeWing;
        MoveL Target_1050,v30,fine,DrillTool\WObj:=FakeWing;
SetDO drillDone,1;
WaitUntil drillDone = 0;
        MoveL RelTool(Target_1050,0,0,-10),v30,z10,DrillTool\WObj:=FakeWing;
        MoveL RelTool(Target_1060,0,0,-10),v30,z10,DrillTool\WObj:=FakeWing;
        MoveL Target_1060,v30,fine,DrillTool\WObj:=FakeWing;
SetDO drillDone,1;
WaitUntil drillDone = 0;
        MoveL RelTool(Target_1060,0,0,-10),v30,z10,DrillTool\WObj:=FakeWing;
        MoveL RelTool(Target_1070,0,0,-10),v30,z10,DrillTool\WObj:=FakeWing;
        MoveL Target_1070,v30,fine,DrillTool\WObj:=FakeWing;
SetDO drillDone,1;
WaitUntil drillDone = 0;
        MoveL RelTool(Target_1070,0,0,-10),v30,z10,DrillTool\WObj:=FakeWing;
        MoveL RelTool(Target_1080,0,0,-10),v30,z10,DrillTool\WObj:=FakeWing;
        MoveL Target_1080,v30,fine,DrillTool\WObj:=FakeWing;
SetDO drillDone,1;
WaitUntil drillDone = 0;
        MoveL RelTool(Target_1080,0,0,-10),v30,z10,DrillTool\WObj:=FakeWing;
        MoveL RelTool(Target_1090,0,0,-10),v30,z10,DrillTool\WObj:=FakeWing;
        MoveL Target_1090,v30,fine,DrillTool\WObj:=FakeWing;
SetDO drillDone,1;
WaitUntil drillDone = 0;
        MoveL RelTool(Target_1090,0,0,-10),v30,z10,DrillTool\WObj:=FakeWing;
        MoveL RelTool(Target_1100,0,0,-10),v30,z10,DrillTool\WObj:=FakeWing;
        MoveL Target_1100,v30,fine,DrillTool\WObj:=FakeWing;
SetDO drillDone,1;
WaitUntil drillDone = 0;
        MoveL RelTool(Target_1100,0,0,-10),v30,z10,DrillTool\WObj:=FakeWing;
        MoveL RelTool(Target_1110,0,0,-10),v30,z10,DrillTool\WObj:=FakeWing;
        MoveL Target_1110,v30,fine,DrillTool\WObj:=FakeWing;
SetDO drillDone,1;
WaitUntil drillDone = 0;
        MoveL RelTool(Target_1110,0,0,-10),v30,z10,DrillTool\WObj:=FakeWing;
        MoveL RelTool(Target_1120,0,0,-10),v30,z10,DrillTool\WObj:=FakeWing;
        MoveL Target_1120,v30,fine,DrillTool\WObj:=FakeWing;
SetDO drillDone,1;
WaitUntil drillDone = 0;
        MoveL RelTool(Target_1120,0,0,-10),v30,z10,DrillTool\WObj:=FakeWing;
        MoveL RelTool(Target_1130,0,0,-10),v30,z10,DrillTool\WObj:=FakeWing;
        MoveL Target_1130,v30,fine,DrillTool\WObj:=FakeWing;
SetDO drillDone,1;
WaitUntil drillDone = 0;
        MoveL RelTool(Target_1130,0,0,-10),v30,z10,DrillTool\WObj:=FakeWing;
        MoveL RelTool(Target_1140,0,0,-10),v30,z10,DrillTool\WObj:=FakeWing;
        MoveL Target_1140,v30,fine,DrillTool\WObj:=FakeWing;
SetDO drillDone,1;
WaitUntil drillDone = 0;
        MoveL RelTool(Target_1140,0,0,-10),v30,z10,DrillTool\WObj:=FakeWing;
        MoveL RelTool(Target_1150,0,0,-10),v30,z10,DrillTool\WObj:=FakeWing;
        MoveL Target_1150,v30,fine,DrillTool\WObj:=FakeWing;
SetDO drillDone,1;
WaitUntil drillDone = 0;
        MoveL RelTool(Target_1150,0,0,-10),v30,z10,DrillTool\WObj:=FakeWing;
        MoveL RelTool(Target_1160,0,0,-10),v30,z10,DrillTool\WObj:=FakeWing;
        MoveL Target_1160,v30,fine,DrillTool\WObj:=FakeWing;
SetDO drillDone,1;
WaitUntil drillDone = 0;
        MoveL RelTool(Target_1160,0,0,-10),v30,z10,DrillTool\WObj:=FakeWing;
        MoveL RelTool(Target_1170,0,0,-10),v30,z10,DrillTool\WObj:=FakeWing;
        MoveL Target_1170,v30,fine,DrillTool\WObj:=FakeWing;
SetDO drillDone,1;
WaitUntil drillDone = 0;
        MoveL RelTool(Target_1170,0,0,-10),v30,z10,DrillTool\WObj:=FakeWing;
        MoveL RelTool(Target_1180,0,0,-10),v30,z10,DrillTool\WObj:=FakeWing;
        MoveL Target_1180,v30,fine,DrillTool\WObj:=FakeWing;
SetDO drillDone,1;
WaitUntil drillDone = 0;
        MoveL RelTool(Target_1180,0,0,-10),v30,z10,DrillTool\WObj:=FakeWing;
        MoveL RelTool(Target_1190,0,0,-10),v30,z10,DrillTool\WObj:=FakeWing;
        MoveL Target_1190,v30,fine,DrillTool\WObj:=FakeWing;
SetDO drillDone,1;
WaitUntil drillDone = 0;
        MoveL RelTool(Target_1190,0,0,-10),v30,z10,DrillTool\WObj:=FakeWing;
        MoveL RelTool(Target_1200,0,0,-10),v30,z10,DrillTool\WObj:=FakeWing;
        MoveL Target_1200,v30,fine,DrillTool\WObj:=FakeWing;
SetDO drillDone,1;
WaitUntil drillDone = 0;
        MoveL RelTool(Target_1200,0,0,-10),v30,z10,DrillTool\WObj:=FakeWing;
        MoveL RelTool(Target_1210,0,0,-10),v30,z10,DrillTool\WObj:=FakeWing;
        MoveL Target_1210,v30,fine,DrillTool\WObj:=FakeWing;
SetDO drillDone,1;
WaitUntil drillDone = 0;
        MoveL RelTool(Target_1210,0,0,-10),v30,z10,DrillTool\WObj:=FakeWing;
        MoveL RelTool(Target_1220,0,0,-10),v30,z10,DrillTool\WObj:=FakeWing;
        MoveL Target_1220,v30,fine,DrillTool\WObj:=FakeWing;
SetDO drillDone,1;
WaitUntil drillDone = 0;
        MoveL RelTool(Target_1220,0,0,-10),v30,z10,DrillTool\WObj:=FakeWing;
        MoveL RelTool(Target_1230,0,0,-10),v30,z10,DrillTool\WObj:=FakeWing;
        MoveL Target_1230,v30,fine,DrillTool\WObj:=FakeWing;
SetDO drillDone,1;
WaitUntil drillDone = 0;
        MoveL RelTool(Target_1230,0,0,-10),v30,z10,DrillTool\WObj:=FakeWing;
        MoveL RelTool(Target_1240,0,0,-10),v30,z10,DrillTool\WObj:=FakeWing;
        MoveL Target_1240,v30,fine,DrillTool\WObj:=FakeWing;
SetDO drillDone,1;
WaitUntil drillDone = 0;
        MoveL RelTool(Target_1240,0,0,-10),v30,z10,DrillTool\WObj:=FakeWing;
        MoveL RelTool(Target_1250,0,0,-10),v30,z10,DrillTool\WObj:=FakeWing;
        MoveL Target_1250,v30,fine,DrillTool\WObj:=FakeWing;
SetDO drillDone,1;
WaitUntil drillDone = 0;
        MoveL RelTool(Target_1250,0,0,-10),v30,z10,DrillTool\WObj:=FakeWing;
        MoveL RelTool(Target_1260,0,0,-10),v30,z10,DrillTool\WObj:=FakeWing;
        MoveL Target_1260,v30,fine,DrillTool\WObj:=FakeWing;
SetDO drillDone,1;
WaitUntil drillDone = 0;
        MoveL RelTool(Target_1260,0,0,-10),v30,z10,DrillTool\WObj:=FakeWing;
        MoveL RelTool(Target_1270,0,0,-10),v30,z10,DrillTool\WObj:=FakeWing;
        MoveL Target_1270,v30,fine,DrillTool\WObj:=FakeWing;
SetDO drillDone,1;
WaitUntil drillDone = 0;
        MoveL RelTool(Target_1270,0,0,-10),v30,z10,DrillTool\WObj:=FakeWing;
        MoveL RelTool(Target_1280,0,0,-10),v30,z10,DrillTool\WObj:=FakeWing;
        MoveL Target_1280,v30,fine,DrillTool\WObj:=FakeWing;
SetDO drillDone,1;
WaitUntil drillDone = 0;
        MoveL RelTool(Target_1280,0,0,-10),v30,z10,DrillTool\WObj:=FakeWing;
        MoveL RelTool(Target_1290,0,0,-10),v30,z10,DrillTool\WObj:=FakeWing;
        MoveL Target_1290,v30,fine,DrillTool\WObj:=FakeWing;
SetDO drillDone,1;
WaitUntil drillDone = 0;
        MoveL RelTool(Target_1290,0,0,-10),v30,z10,DrillTool\WObj:=FakeWing;
        MoveL RelTool(Target_1300,0,0,-10),v30,z10,DrillTool\WObj:=FakeWing;
        MoveL Target_1300,v30,fine,DrillTool\WObj:=FakeWing;
SetDO drillDone,1;
WaitUntil drillDone = 0;
        MoveL RelTool(Target_1300,0,0,-10),v30,z10,DrillTool\WObj:=FakeWing;
        MoveL RelTool(Target_1310,0,0,-10),v30,z10,DrillTool\WObj:=FakeWing;
        MoveL Target_1310,v30,fine,DrillTool\WObj:=FakeWing;
SetDO drillDone,1;
WaitUntil drillDone = 0;
        MoveL RelTool(Target_1310,0,0,-10),v30,z10,DrillTool\WObj:=FakeWing;
        MoveL RelTool(Target_1320,0,0,-10),v30,z10,DrillTool\WObj:=FakeWing;
        MoveL Target_1320,v30,fine,DrillTool\WObj:=FakeWing;
SetDO drillDone,1;
WaitUntil drillDone = 0;
        MoveL RelTool(Target_1320,0,0,-10),v30,z10,DrillTool\WObj:=FakeWing;
        MoveL RelTool(Target_1330,0,0,-10),v30,z10,DrillTool\WObj:=FakeWing;
        MoveL Target_1330,v30,fine,DrillTool\WObj:=FakeWing;
SetDO drillDone,1;
WaitUntil drillDone = 0;
        MoveL RelTool(Target_1330,0,0,-10),v30,z10,DrillTool\WObj:=FakeWing;
        MoveL RelTool(Target_1340,0,0,-10),v30,z10,DrillTool\WObj:=FakeWing;
        MoveL Target_1340,v30,fine,DrillTool\WObj:=FakeWing;
SetDO drillDone,1;
WaitUntil drillDone = 0;
        MoveL RelTool(Target_1340,0,0,-10),v30,z10,DrillTool\WObj:=FakeWing;
        MoveL RelTool(Target_1350,0,0,-10),v30,z10,DrillTool\WObj:=FakeWing;
        MoveL Target_1350,v30,fine,DrillTool\WObj:=FakeWing;
SetDO drillDone,1;
WaitUntil drillDone = 0;
        MoveL RelTool(Target_1350,0,0,-10),v30,z10,DrillTool\WObj:=FakeWing;
        MoveL RelTool(Target_1360,0,0,-10),v30,z10,DrillTool\WObj:=FakeWing;
        MoveL Target_1360,v30,fine,DrillTool\WObj:=FakeWing;
SetDO drillDone,1;
WaitUntil drillDone = 0;
        MoveL RelTool(Target_1360,0,0,-10),v30,z10,DrillTool\WObj:=FakeWing;
        MoveL RelTool(Target_1370,0,0,-10),v30,z10,DrillTool\WObj:=FakeWing;
        MoveL Target_1370,v30,fine,DrillTool\WObj:=FakeWing;
SetDO drillDone,1;
WaitUntil drillDone = 0;
        MoveL RelTool(Target_1370,0,0,-10),v30,z10,DrillTool\WObj:=FakeWing;
        MoveL RelTool(Target_1380,0,0,-10),v30,z10,DrillTool\WObj:=FakeWing;
        MoveL Target_1380,v30,fine,DrillTool\WObj:=FakeWing;
SetDO drillDone,1;
WaitUntil drillDone = 0;
        MoveL RelTool(Target_1380,0,0,-10),v30,z10,DrillTool\WObj:=FakeWing;
        MoveL RelTool(Target_1390,0,0,-10),v30,z10,DrillTool\WObj:=FakeWing;
        MoveL Target_1390,v30,fine,DrillTool\WObj:=FakeWing;
SetDO drillDone,1;
WaitUntil drillDone = 0;
        MoveL RelTool(Target_1390,0,0,-10),v30,z10,DrillTool\WObj:=FakeWing;
        MoveL RelTool(Target_1400,0,0,-10),v30,z10,DrillTool\WObj:=FakeWing;
        MoveL Target_1400,v30,fine,DrillTool\WObj:=FakeWing;
SetDO drillDone,1;
WaitUntil drillDone = 0;
        MoveL RelTool(Target_1400,0,0,-10),v30,z10,DrillTool\WObj:=FakeWing;
        MoveL RelTool(Target_1410,0,0,-10),v30,z10,DrillTool\WObj:=FakeWing;
        MoveL Target_1410,v30,fine,DrillTool\WObj:=FakeWing;
SetDO drillDone,1;
WaitUntil drillDone = 0;
        MoveL RelTool(Target_1410,0,0,-10),v30,z10,DrillTool\WObj:=FakeWing;
        MoveL RelTool(Target_1420,0,0,-10),v30,z10,DrillTool\WObj:=FakeWing;
        MoveL Target_1420,v30,fine,DrillTool\WObj:=FakeWing;
SetDO drillDone,1;
WaitUntil drillDone = 0;
        MoveL RelTool(Target_1420,0,0,-10),v30,z10,DrillTool\WObj:=FakeWing;
        MoveL RelTool(Target_1430,0,0,-10),v30,z10,DrillTool\WObj:=FakeWing;
        MoveL Target_1430,v30,fine,DrillTool\WObj:=FakeWing;
SetDO drillDone,1;
WaitUntil drillDone = 0;
        MoveL RelTool(Target_1430,0,0,-10),v30,z10,DrillTool\WObj:=FakeWing;
        MoveL RelTool(Target_1440,0,0,-10),v30,z10,DrillTool\WObj:=FakeWing;
        MoveL Target_1440,v30,fine,DrillTool\WObj:=FakeWing;
SetDO drillDone,1;
WaitUntil drillDone = 0;
        MoveL RelTool(Target_1440,0,0,-10),v30,z10,DrillTool\WObj:=FakeWing;
        MoveL RelTool(Target_1450,0,0,-10),v30,z10,DrillTool\WObj:=FakeWing;
        MoveL Target_1450,v30,fine,DrillTool\WObj:=FakeWing;
SetDO drillDone,1;
WaitUntil drillDone = 0;
        MoveL RelTool(Target_1450,0,0,-10),v30,z10,DrillTool\WObj:=FakeWing;
        MoveL RelTool(Target_1460,0,0,-10),v30,z10,DrillTool\WObj:=FakeWing;
        MoveL Target_1460,v30,fine,DrillTool\WObj:=FakeWing;
SetDO drillDone,1;
WaitUntil drillDone = 0;
        MoveL RelTool(Target_1460,0,0,-10),v30,z10,DrillTool\WObj:=FakeWing;
        MoveL RelTool(Target_1470,0,0,-10),v30,z10,DrillTool\WObj:=FakeWing;
        MoveL Target_1470,v30,fine,DrillTool\WObj:=FakeWing;
SetDO drillDone,1;
WaitUntil drillDone = 0;
        MoveL RelTool(Target_1470,0,0,-10),v30,z10,DrillTool\WObj:=FakeWing;
        MoveL RelTool(Target_1480,0,0,-10),v30,z10,DrillTool\WObj:=FakeWing;
        MoveL Target_1480,v30,fine,DrillTool\WObj:=FakeWing;
SetDO drillDone,1;
WaitUntil drillDone = 0;
        MoveL RelTool(Target_1480,0,0,-10),v30,z10,DrillTool\WObj:=FakeWing;
        MoveL RelTool(Target_1490,0,0,-10),v30,z10,DrillTool\WObj:=FakeWing;
        MoveL Target_1490,v30,fine,DrillTool\WObj:=FakeWing;
SetDO drillDone,1;
WaitUntil drillDone = 0;
        MoveL RelTool(Target_1490,0,0,-10),v30,z10,DrillTool\WObj:=FakeWing;
        MoveL RelTool(Target_1500,0,0,-10),v30,z10,DrillTool\WObj:=FakeWing;
        MoveL Target_1500,v30,fine,DrillTool\WObj:=FakeWing;
SetDO drillDone,1;
WaitUntil drillDone = 0;
        MoveL RelTool(Target_1500,0,0,-10),v30,z10,DrillTool\WObj:=FakeWing;
        MoveL RelTool(Target_1510,0,0,-10),v30,z10,DrillTool\WObj:=FakeWing;
        MoveL Target_1510,v30,fine,DrillTool\WObj:=FakeWing;
SetDO drillDone,1;
WaitUntil drillDone = 0;
        MoveL RelTool(Target_1510,0,0,-10),v30,z10,DrillTool\WObj:=FakeWing;
        MoveL RelTool(Target_1520,0,0,-10),v30,z10,DrillTool\WObj:=FakeWing;
        MoveL Target_1520,v30,fine,DrillTool\WObj:=FakeWing;
SetDO drillDone,1;
WaitUntil drillDone = 0;
        MoveL RelTool(Target_1520,0,0,-10),v30,z10,DrillTool\WObj:=FakeWing;
        MoveL RelTool(Target_1530,0,0,-10),v30,z10,DrillTool\WObj:=FakeWing;
        MoveL Target_1530,v30,fine,DrillTool\WObj:=FakeWing;
SetDO drillDone,1;
WaitUntil drillDone = 0;
        MoveL RelTool(Target_1530,0,0,-10),v30,z10,DrillTool\WObj:=FakeWing;
        MoveL RelTool(Target_1540,0,0,-10),v30,z10,DrillTool\WObj:=FakeWing;
        MoveL Target_1540,v30,fine,DrillTool\WObj:=FakeWing;
SetDO drillDone,1;
WaitUntil drillDone = 0;
        MoveL RelTool(Target_1540,0,0,-10),v30,z10,DrillTool\WObj:=FakeWing;
        MoveL RelTool(Target_1550,0,0,-10),v30,z10,DrillTool\WObj:=FakeWing;
        MoveL Target_1550,v30,fine,DrillTool\WObj:=FakeWing;
SetDO drillDone,1;
WaitUntil drillDone = 0;
        MoveL RelTool(Target_1550,0,0,-10),v30,z10,DrillTool\WObj:=FakeWing;
        MoveL RelTool(Target_1560,0,0,-10),v30,z10,DrillTool\WObj:=FakeWing;
        MoveL Target_1560,v30,fine,DrillTool\WObj:=FakeWing;
SetDO drillDone,1;
WaitUntil drillDone = 0;
        MoveL RelTool(Target_1560,0,0,-10),v30,z10,DrillTool\WObj:=FakeWing;
        MoveL RelTool(Target_1570,0,0,-10),v30,z10,DrillTool\WObj:=FakeWing;
        MoveL Target_1570,v30,fine,DrillTool\WObj:=FakeWing;
SetDO drillDone,1;
WaitUntil drillDone = 0;
        MoveL RelTool(Target_1570,0,0,-10),v30,z10,DrillTool\WObj:=FakeWing;
        MoveL RelTool(Target_1580,0,0,-10),v30,z10,DrillTool\WObj:=FakeWing;
        MoveL Target_1580,v30,fine,DrillTool\WObj:=FakeWing;
SetDO drillDone,1;
WaitUntil drillDone = 0;
        MoveL RelTool(Target_1580,0,0,-10),v30,z10,DrillTool\WObj:=FakeWing;
        MoveL RelTool(Target_1590,0,0,-10),v30,z10,DrillTool\WObj:=FakeWing;
        MoveL Target_1590,v30,fine,DrillTool\WObj:=FakeWing;
SetDO drillDone,1;
WaitUntil drillDone = 0;
        MoveL RelTool(Target_1590,0,0,-10),v30,z10,DrillTool\WObj:=FakeWing;
        MoveL RelTool(Target_1600,0,0,-10),v30,z10,DrillTool\WObj:=FakeWing;
        MoveL Target_1600,v30,fine,DrillTool\WObj:=FakeWing;
SetDO drillDone,1;
WaitUntil drillDone = 0;
        MoveL RelTool(Target_1600,0,0,-10),v30,z10,DrillTool\WObj:=FakeWing;
        MoveL RelTool(Target_1610,0,0,-10),v30,z10,DrillTool\WObj:=FakeWing;
        MoveL Target_1610,v30,fine,DrillTool\WObj:=FakeWing;
SetDO drillDone,1;
WaitUntil drillDone = 0;
        MoveL RelTool(Target_1610,0,0,-10),v30,z10,DrillTool\WObj:=FakeWing;
        MoveL RelTool(Target_1620,0,0,-10),v30,z10,DrillTool\WObj:=FakeWing;
        MoveL Target_1620,v30,fine,DrillTool\WObj:=FakeWing;
SetDO drillDone,1;
WaitUntil drillDone = 0;
        MoveL RelTool(Target_1620,0,0,-10),v30,z10,DrillTool\WObj:=FakeWing;
        MoveL RelTool(Target_1630,0,0,-10),v30,z10,DrillTool\WObj:=FakeWing;
        MoveL Target_1630,v30,fine,DrillTool\WObj:=FakeWing;
SetDO drillDone,1;
WaitUntil drillDone = 0;
        MoveL RelTool(Target_1630,0,0,-10),v30,z10,DrillTool\WObj:=FakeWing;
        MoveL RelTool(Target_1640,0,0,-10),v30,z10,DrillTool\WObj:=FakeWing;
        MoveL Target_1640,v30,fine,DrillTool\WObj:=FakeWing;
SetDO drillDone,1;
WaitUntil drillDone = 0;
        MoveL RelTool(Target_1640,0,0,-10),v30,z10,DrillTool\WObj:=FakeWing;
        MoveL RelTool(Target_1650,0,0,-10),v30,z10,DrillTool\WObj:=FakeWing;
        MoveL Target_1650,v30,fine,DrillTool\WObj:=FakeWing;
SetDO drillDone,1;
WaitUntil drillDone = 0;
        MoveL RelTool(Target_1650,0,0,-10),v30,z10,DrillTool\WObj:=FakeWing;
        MoveL RelTool(Target_1660,0,0,-10),v30,z10,DrillTool\WObj:=FakeWing;
        MoveL Target_1660,v30,fine,DrillTool\WObj:=FakeWing;
SetDO drillDone,1;
WaitUntil drillDone = 0;
        MoveL RelTool(Target_1660,0,0,-10),v30,z10,DrillTool\WObj:=FakeWing;
        MoveL RelTool(Target_1670,0,0,-10),v30,z10,DrillTool\WObj:=FakeWing;
        MoveL Target_1670,v30,fine,DrillTool\WObj:=FakeWing;
SetDO drillDone,1;
WaitUntil drillDone = 0;
        MoveL RelTool(Target_1670,0,0,-10),v30,z10,DrillTool\WObj:=FakeWing;
        MoveL RelTool(Target_1680,0,0,-10),v30,z10,DrillTool\WObj:=FakeWing;
        MoveL Target_1680,v30,fine,DrillTool\WObj:=FakeWing;
SetDO drillDone,1;
WaitUntil drillDone = 0;
        MoveL RelTool(Target_1680,0,0,-10),v30,z10,DrillTool\WObj:=FakeWing;
        MoveL RelTool(Target_1690,0,0,-10),v30,z10,DrillTool\WObj:=FakeWing;
        MoveL Target_1690,v30,fine,DrillTool\WObj:=FakeWing;
SetDO drillDone,1;
WaitUntil drillDone = 0;
        MoveL RelTool(Target_1690,0,0,-10),v30,z10,DrillTool\WObj:=FakeWing;
        MoveL RelTool(Target_1700,0,0,-10),v30,z10,DrillTool\WObj:=FakeWing;
        MoveL Target_1700,v30,fine,DrillTool\WObj:=FakeWing;
SetDO drillDone,1;
WaitUntil drillDone = 0;
        MoveL RelTool(Target_1700,0,0,-10),v30,z10,DrillTool\WObj:=FakeWing;
        MoveL RelTool(Target_1710,0,0,-10),v30,z10,DrillTool\WObj:=FakeWing;
        MoveL Target_1710,v30,fine,DrillTool\WObj:=FakeWing;
SetDO drillDone,1;
WaitUntil drillDone = 0;
        MoveL RelTool(Target_1710,0,0,-10),v30,z10,DrillTool\WObj:=FakeWing;
        MoveL RelTool(Target_1720,0,0,-10),v30,z10,DrillTool\WObj:=FakeWing;
        MoveL Target_1720,v30,fine,DrillTool\WObj:=FakeWing;
SetDO drillDone,1;
WaitUntil drillDone = 0;
        MoveL RelTool(Target_1720,0,0,-10),v30,z10,DrillTool\WObj:=FakeWing;
        MoveL RelTool(Target_1730,0,0,-10),v30,z10,DrillTool\WObj:=FakeWing;
        MoveL Target_1730,v30,fine,DrillTool\WObj:=FakeWing;
SetDO drillDone,1;
WaitUntil drillDone = 0;
        MoveL RelTool(Target_1730,0,0,-10),v30,z10,DrillTool\WObj:=FakeWing;
        MoveL RelTool(Target_1740,0,0,-10),v30,z10,DrillTool\WObj:=FakeWing;
        MoveL Target_1740,v30,fine,DrillTool\WObj:=FakeWing;
SetDO drillDone,1;
WaitUntil drillDone = 0;
        MoveL RelTool(Target_1740,0,0,-10),v30,z10,DrillTool\WObj:=FakeWing;
        MoveL RelTool(Target_1750,0,0,-10),v30,z10,DrillTool\WObj:=FakeWing;
        MoveL Target_1750,v30,fine,DrillTool\WObj:=FakeWing;
SetDO drillDone,1;
WaitUntil drillDone = 0;
        MoveL RelTool(Target_1750,0,0,-10),v30,z10,DrillTool\WObj:=FakeWing;
        MoveL RelTool(Target_1760,0,0,-10),v30,z10,DrillTool\WObj:=FakeWing;
        MoveL Target_1760,v30,fine,DrillTool\WObj:=FakeWing;
SetDO drillDone,1;
WaitUntil drillDone = 0;
        MoveL RelTool(Target_1760,0,0,-10),v30,z10,DrillTool\WObj:=FakeWing;
        MoveL RelTool(Target_1770,0,0,-10),v30,z10,DrillTool\WObj:=FakeWing;
        MoveL Target_1770,v30,fine,DrillTool\WObj:=FakeWing;
SetDO drillDone,1;
WaitUntil drillDone = 0;
        MoveL RelTool(Target_1770,0,0,-10),v30,z10,DrillTool\WObj:=FakeWing;
        MoveL RelTool(Target_1780,0,0,-10),v30,z10,DrillTool\WObj:=FakeWing;
        MoveL Target_1780,v30,fine,DrillTool\WObj:=FakeWing;
SetDO drillDone,1;
WaitUntil drillDone = 0;
        MoveL RelTool(Target_1780,0,0,-10),v30,z10,DrillTool\WObj:=FakeWing;
        MoveL RelTool(Target_1790,0,0,-10),v30,z10,DrillTool\WObj:=FakeWing;
        MoveL Target_1790,v30,fine,DrillTool\WObj:=FakeWing;
SetDO drillDone,1;
WaitUntil drillDone = 0;
        MoveL RelTool(Target_1790,0,0,-10),v30,z10,DrillTool\WObj:=FakeWing;
        MoveL RelTool(Target_1800,0,0,-10),v30,z10,DrillTool\WObj:=FakeWing;
        MoveL Target_1800,v30,fine,DrillTool\WObj:=FakeWing;
SetDO drillDone,1;
WaitUntil drillDone = 0;
        MoveL RelTool(Target_1800,0,0,-10),v30,z10,DrillTool\WObj:=FakeWing;
        MoveL RelTool(Target_1810,0,0,-10),v30,z10,DrillTool\WObj:=FakeWing;
        MoveL Target_1810,v30,fine,DrillTool\WObj:=FakeWing;
SetDO drillDone,1;
WaitUntil drillDone = 0;
        MoveL RelTool(Target_1810,0,0,-10),v30,z10,DrillTool\WObj:=FakeWing;
        MoveL RelTool(Target_1820,0,0,-10),v30,z10,DrillTool\WObj:=FakeWing;
        MoveL Target_1820,v30,fine,DrillTool\WObj:=FakeWing;
SetDO drillDone,1;
WaitUntil drillDone = 0;
        MoveL RelTool(Target_1820,0,0,-10),v30,z10,DrillTool\WObj:=FakeWing;
        MoveL RelTool(Target_1830,0,0,-10),v30,z10,DrillTool\WObj:=FakeWing;
        MoveL Target_1830,v30,fine,DrillTool\WObj:=FakeWing;
SetDO drillDone,1;
WaitUntil drillDone = 0;
        MoveL RelTool(Target_1830,0,0,-10),v30,z10,DrillTool\WObj:=FakeWing;
        MoveL RelTool(Target_1840,0,0,-10),v30,z10,DrillTool\WObj:=FakeWing;
        MoveL Target_1840,v30,fine,DrillTool\WObj:=FakeWing;
SetDO drillDone,1;
WaitUntil drillDone = 0;
        MoveL RelTool(Target_1840,0,0,-10),v30,z10,DrillTool\WObj:=FakeWing;
        MoveL RelTool(Target_1850,0,0,-10),v30,z10,DrillTool\WObj:=FakeWing;
        MoveL Target_1850,v30,fine,DrillTool\WObj:=FakeWing;
SetDO drillDone,1;
WaitUntil drillDone = 0;
        MoveL RelTool(Target_1850,0,0,-10),v30,z10,DrillTool\WObj:=FakeWing;
        MoveL RelTool(Target_1860,0,0,-10),v30,z10,DrillTool\WObj:=FakeWing;
        MoveL Target_1860,v30,fine,DrillTool\WObj:=FakeWing;
SetDO drillDone,1;
WaitUntil drillDone = 0;
        MoveL RelTool(Target_1860,0,0,-10),v30,z10,DrillTool\WObj:=FakeWing;
        MoveL RelTool(Target_1870,0,0,-10),v30,z10,DrillTool\WObj:=FakeWing;
        MoveL Target_1870,v30,fine,DrillTool\WObj:=FakeWing;
SetDO drillDone,1;
WaitUntil drillDone = 0;
        MoveL RelTool(Target_1870,0,0,-10),v30,z10,DrillTool\WObj:=FakeWing;
        MoveL RelTool(Target_1880,0,0,-10),v30,z10,DrillTool\WObj:=FakeWing;
        MoveL Target_1880,v30,fine,DrillTool\WObj:=FakeWing;
SetDO drillDone,1;
WaitUntil drillDone = 0;
        MoveL RelTool(Target_1880,0,0,-10),v30,z10,DrillTool\WObj:=FakeWing;
        MoveL RelTool(Target_1890,0,0,-10),v30,z10,DrillTool\WObj:=FakeWing;
        MoveL Target_1890,v30,fine,DrillTool\WObj:=FakeWing;
SetDO drillDone,1;
WaitUntil drillDone = 0;
        MoveL RelTool(Target_1890,0,0,-10),v30,z10,DrillTool\WObj:=FakeWing;
        MoveL RelTool(Target_1900,0,0,-10),v30,z10,DrillTool\WObj:=FakeWing;
        MoveL Target_1900,v30,fine,DrillTool\WObj:=FakeWing;
SetDO drillDone,1;
WaitUntil drillDone = 0;
        MoveL RelTool(Target_1900,0,0,-10),v30,z10,DrillTool\WObj:=FakeWing;
        MoveL RelTool(Target_1910,0,0,-10),v30,z10,DrillTool\WObj:=FakeWing;
        MoveL Target_1910,v30,fine,DrillTool\WObj:=FakeWing;
SetDO drillDone,1;
WaitUntil drillDone = 0;
        MoveL RelTool(Target_1910,0,0,-10),v30,z10,DrillTool\WObj:=FakeWing;
        MoveL RelTool(Target_1920,0,0,-10),v30,z10,DrillTool\WObj:=FakeWing;
        MoveL Target_1920,v30,fine,DrillTool\WObj:=FakeWing;
SetDO drillDone,1;
WaitUntil drillDone = 0;
        MoveL RelTool(Target_1920,0,0,-10),v30,z10,DrillTool\WObj:=FakeWing;
        MoveL RelTool(Target_1930,0,0,-10),v30,z10,DrillTool\WObj:=FakeWing;
        MoveL Target_1930,v30,fine,DrillTool\WObj:=FakeWing;
SetDO drillDone,1;
WaitUntil drillDone = 0;
        MoveL RelTool(Target_1930,0,0,-10),v30,z10,DrillTool\WObj:=FakeWing;
        MoveL RelTool(Target_1940,0,0,-10),v30,z10,DrillTool\WObj:=FakeWing;
        MoveL Target_1940,v30,fine,DrillTool\WObj:=FakeWing;
SetDO drillDone,1;
WaitUntil drillDone = 0;
        MoveL RelTool(Target_1940,0,0,-10),v30,z10,DrillTool\WObj:=FakeWing;
        MoveL RelTool(Target_1950,0,0,-10),v30,z10,DrillTool\WObj:=FakeWing;
        MoveL Target_1950,v30,fine,DrillTool\WObj:=FakeWing;
SetDO drillDone,1;
WaitUntil drillDone = 0;
        MoveL RelTool(Target_1950,0,0,-10),v30,z10,DrillTool\WObj:=FakeWing;
        MoveL RelTool(Target_1960,0,0,-10),v30,z10,DrillTool\WObj:=FakeWing;
        MoveL Target_1960,v30,fine,DrillTool\WObj:=FakeWing;
SetDO drillDone,1;
WaitUntil drillDone = 0;
        MoveL RelTool(Target_1960,0,0,-10),v30,z10,DrillTool\WObj:=FakeWing;
        MoveL RelTool(Target_1970,0,0,-10),v30,z10,DrillTool\WObj:=FakeWing;
        MoveL Target_1970,v30,fine,DrillTool\WObj:=FakeWing;
SetDO drillDone,1;
WaitUntil drillDone = 0;
        MoveL RelTool(Target_1970,0,0,-10),v30,z10,DrillTool\WObj:=FakeWing;
        MoveL RelTool(Target_1980,0,0,-10),v30,z10,DrillTool\WObj:=FakeWing;
        MoveL Target_1980,v30,fine,DrillTool\WObj:=FakeWing;
SetDO drillDone,1;
WaitUntil drillDone = 0;
        MoveL RelTool(Target_1980,0,0,-10),v30,z10,DrillTool\WObj:=FakeWing;
        MoveL RelTool(Target_1990,0,0,-10),v30,z10,DrillTool\WObj:=FakeWing;
        MoveL Target_1990,v30,fine,DrillTool\WObj:=FakeWing;
SetDO drillDone,1;
WaitUntil drillDone = 0;
        MoveL RelTool(Target_1990,0,0,-10),v30,z10,DrillTool\WObj:=FakeWing;
        MoveL RelTool(Target_2000,0,0,-10),v30,z10,DrillTool\WObj:=FakeWing;
        MoveL Target_2000,v30,fine,DrillTool\WObj:=FakeWing;
SetDO drillDone,1;
WaitUntil drillDone = 0;
        MoveL RelTool(Target_2000,0,0,-10),v30,z10,DrillTool\WObj:=FakeWing;
        MoveL RelTool(Target_2010,0,0,-10),v30,z10,DrillTool\WObj:=FakeWing;
        MoveL Target_2010,v30,fine,DrillTool\WObj:=FakeWing;
SetDO drillDone,1;
WaitUntil drillDone = 0;
        MoveL RelTool(Target_2010,0,0,-10),v30,z10,DrillTool\WObj:=FakeWing;
        MoveL RelTool(Target_2020,0,0,-10),v30,z10,DrillTool\WObj:=FakeWing;
        MoveL Target_2020,v30,fine,DrillTool\WObj:=FakeWing;
SetDO drillDone,1;
WaitUntil drillDone = 0;
        MoveL RelTool(Target_2020,0,0,-10),v30,z10,DrillTool\WObj:=FakeWing;
        MoveL RelTool(Target_2030,0,0,-10),v30,z10,DrillTool\WObj:=FakeWing;
        MoveL Target_2030,v30,fine,DrillTool\WObj:=FakeWing;
SetDO drillDone,1;
WaitUntil drillDone = 0;
        MoveL RelTool(Target_2030,0,0,-10),v30,z10,DrillTool\WObj:=FakeWing;
        MoveL RelTool(Target_2040,0,0,-10),v30,z10,DrillTool\WObj:=FakeWing;
        MoveL Target_2040,v30,fine,DrillTool\WObj:=FakeWing;
SetDO drillDone,1;
WaitUntil drillDone = 0;
        MoveL RelTool(Target_2040,0,0,-10),v30,z10,DrillTool\WObj:=FakeWing;
        MoveL RelTool(Target_2050,0,0,-10),v30,z10,DrillTool\WObj:=FakeWing;
        MoveL Target_2050,v30,fine,DrillTool\WObj:=FakeWing;
SetDO drillDone,1;
WaitUntil drillDone = 0;
        MoveL RelTool(Target_2050,0,0,-10),v30,z10,DrillTool\WObj:=FakeWing;
        MoveL RelTool(Target_2060,0,0,-10),v30,z10,DrillTool\WObj:=FakeWing;
        MoveL Target_2060,v30,fine,DrillTool\WObj:=FakeWing;
SetDO drillDone,1;
WaitUntil drillDone = 0;
        MoveL RelTool(Target_2060,0,0,-10),v30,z10,DrillTool\WObj:=FakeWing;
        MoveL RelTool(Target_2070,0,0,-10),v30,z10,DrillTool\WObj:=FakeWing;
        MoveL Target_2070,v30,fine,DrillTool\WObj:=FakeWing;
SetDO drillDone,1;
WaitUntil drillDone = 0;
        MoveL RelTool(Target_2070,0,0,-10),v30,z10,DrillTool\WObj:=FakeWing;
        MoveL RelTool(Target_2080,0,0,-10),v30,z10,DrillTool\WObj:=FakeWing;
        MoveL Target_2080,v30,fine,DrillTool\WObj:=FakeWing;
SetDO drillDone,1;
WaitUntil drillDone = 0;
        MoveL RelTool(Target_2080,0,0,-10),v30,z10,DrillTool\WObj:=FakeWing;
        MoveL RelTool(Target_2090,0,0,-10),v30,z10,DrillTool\WObj:=FakeWing;
        MoveL Target_2090,v30,fine,DrillTool\WObj:=FakeWing;
SetDO drillDone,1;
WaitUntil drillDone = 0;
        MoveL RelTool(Target_2090,0,0,-10),v30,z10,DrillTool\WObj:=FakeWing;
        MoveL RelTool(Target_2100,0,0,-10),v30,z10,DrillTool\WObj:=FakeWing;
        MoveL Target_2100,v30,fine,DrillTool\WObj:=FakeWing;
SetDO drillDone,1;
WaitUntil drillDone = 0;
        MoveL RelTool(Target_2100,0,0,-10),v30,z10,DrillTool\WObj:=FakeWing;
        MoveL RelTool(Target_2110,0,0,-10),v30,z10,DrillTool\WObj:=FakeWing;
        MoveL Target_2110,v30,fine,DrillTool\WObj:=FakeWing;
SetDO drillDone,1;
WaitUntil drillDone = 0;
        MoveL RelTool(Target_2110,0,0,-10),v30,z10,DrillTool\WObj:=FakeWing;
        MoveL RelTool(Target_2120,0,0,-10),v30,z10,DrillTool\WObj:=FakeWing;
        MoveL Target_2120,v30,fine,DrillTool\WObj:=FakeWing;
SetDO drillDone,1;
WaitUntil drillDone = 0;
        MoveL RelTool(Target_2120,0,0,-10),v30,z10,DrillTool\WObj:=FakeWing;
        MoveL RelTool(Target_2130,0,0,-10),v30,z10,DrillTool\WObj:=FakeWing;
        MoveL Target_2130,v30,fine,DrillTool\WObj:=FakeWing;
SetDO drillDone,1;
WaitUntil drillDone = 0;
        MoveL RelTool(Target_2130,0,0,-10),v30,z10,DrillTool\WObj:=FakeWing;
        MoveL RelTool(Target_2140,0,0,-10),v30,z10,DrillTool\WObj:=FakeWing;
        MoveL Target_2140,v30,fine,DrillTool\WObj:=FakeWing;
SetDO drillDone,1;
WaitUntil drillDone = 0;
        MoveL RelTool(Target_2140,0,0,-10),v30,z10,DrillTool\WObj:=FakeWing;
        MoveL RelTool(Target_2150,0,0,-10),v30,z10,DrillTool\WObj:=FakeWing;
        MoveL Target_2150,v30,fine,DrillTool\WObj:=FakeWing;
SetDO drillDone,1;
WaitUntil drillDone = 0;
        MoveL RelTool(Target_2150,0,0,-10),v30,z10,DrillTool\WObj:=FakeWing;
        MoveL RelTool(Target_2160,0,0,-10),v30,z10,DrillTool\WObj:=FakeWing;
        MoveL Target_2160,v30,fine,DrillTool\WObj:=FakeWing;
SetDO drillDone,1;
WaitUntil drillDone = 0;
        MoveL RelTool(Target_2160,0,0,-10),v30,z10,DrillTool\WObj:=FakeWing;
        MoveL RelTool(Target_2170,0,0,-10),v30,z10,DrillTool\WObj:=FakeWing;
        MoveL Target_2170,v30,fine,DrillTool\WObj:=FakeWing;
SetDO drillDone,1;
WaitUntil drillDone = 0;
        MoveL RelTool(Target_2170,0,0,-10),v30,z10,DrillTool\WObj:=FakeWing;
        MoveL RelTool(Target_2180,0,0,-10),v30,z10,DrillTool\WObj:=FakeWing;
        MoveL Target_2180,v30,fine,DrillTool\WObj:=FakeWing;
SetDO drillDone,1;
WaitUntil drillDone = 0;
        MoveL RelTool(Target_2180,0,0,-10),v30,z10,DrillTool\WObj:=FakeWing;
        MoveL RelTool(Target_2190,0,0,-10),v30,z10,DrillTool\WObj:=FakeWing;
        MoveL Target_2190,v30,fine,DrillTool\WObj:=FakeWing;
SetDO drillDone,1;
WaitUntil drillDone = 0;
        MoveL RelTool(Target_2190,0,0,-10),v30,z10,DrillTool\WObj:=FakeWing;
        MoveL RelTool(Target_2200,0,0,-10),v30,z10,DrillTool\WObj:=FakeWing;
        MoveL Target_2200,v30,fine,DrillTool\WObj:=FakeWing;
SetDO drillDone,1;
WaitUntil drillDone = 0;
        MoveL RelTool(Target_2200,0,0,-10),v30,z10,DrillTool\WObj:=FakeWing;
        MoveL RelTool(Target_2210,0,0,-10),v30,z10,DrillTool\WObj:=FakeWing;
        MoveL Target_2210,v30,fine,DrillTool\WObj:=FakeWing;
SetDO drillDone,1;
WaitUntil drillDone = 0;
        MoveL RelTool(Target_2210,0,0,-10),v30,z10,DrillTool\WObj:=FakeWing;
        MoveL RelTool(Target_2220,0,0,-10),v30,z10,DrillTool\WObj:=FakeWing;
        MoveL Target_2220,v30,fine,DrillTool\WObj:=FakeWing;
SetDO drillDone,1;
WaitUntil drillDone = 0;
        MoveL RelTool(Target_2220,0,0,-10),v30,z10,DrillTool\WObj:=FakeWing;
        MoveL RelTool(Target_2230,0,0,-10),v30,z10,DrillTool\WObj:=FakeWing;
        MoveL Target_2230,v30,fine,DrillTool\WObj:=FakeWing;
SetDO drillDone,1;
WaitUntil drillDone = 0;
        MoveL RelTool(Target_2230,0,0,-10),v30,z10,DrillTool\WObj:=FakeWing;
        MoveL RelTool(Target_2240,0,0,-10),v30,z10,DrillTool\WObj:=FakeWing;
        MoveL Target_2240,v30,fine,DrillTool\WObj:=FakeWing;
SetDO drillDone,1;
WaitUntil drillDone = 0;
        MoveL RelTool(Target_2240,0,0,-10),v30,z10,DrillTool\WObj:=FakeWing;
        MoveL RelTool(Target_2250,0,0,-10),v30,z10,DrillTool\WObj:=FakeWing;
        MoveL Target_2250,v30,fine,DrillTool\WObj:=FakeWing;
SetDO drillDone,1;
WaitUntil drillDone = 0;
        MoveL RelTool(Target_2250,0,0,-10),v30,z10,DrillTool\WObj:=FakeWing;
        MoveL RelTool(Target_2260,0,0,-10),v30,z10,DrillTool\WObj:=FakeWing;
        MoveL Target_2260,v30,fine,DrillTool\WObj:=FakeWing;
SetDO drillDone,1;
WaitUntil drillDone = 0;
        MoveL RelTool(Target_2260,0,0,-10),v30,z10,DrillTool\WObj:=FakeWing;
        MoveL RelTool(Target_2270,0,0,-10),v30,z10,DrillTool\WObj:=FakeWing;
        MoveL Target_2270,v30,fine,DrillTool\WObj:=FakeWing;
SetDO drillDone,1;
WaitUntil drillDone = 0;
        MoveL RelTool(Target_2270,0,0,-10),v30,z10,DrillTool\WObj:=FakeWing;
        MoveL RelTool(Target_2280,0,0,-10),v30,z10,DrillTool\WObj:=FakeWing;
        MoveL Target_2280,v30,fine,DrillTool\WObj:=FakeWing;
SetDO drillDone,1;
WaitUntil drillDone = 0;
        MoveL RelTool(Target_2280,0,0,-10),v30,z10,DrillTool\WObj:=FakeWing;
        MoveL RelTool(Target_2290,0,0,-10),v30,z10,DrillTool\WObj:=FakeWing;
        MoveL Target_2290,v30,fine,DrillTool\WObj:=FakeWing;
SetDO drillDone,1;
WaitUntil drillDone = 0;
        MoveL RelTool(Target_2290,0,0,-10),v30,z10,DrillTool\WObj:=FakeWing;
        MoveL RelTool(Target_2300,0,0,-10),v30,z10,DrillTool\WObj:=FakeWing;
        MoveL Target_2300,v30,fine,DrillTool\WObj:=FakeWing;
SetDO drillDone,1;
WaitUntil drillDone = 0;
        MoveL RelTool(Target_2300,0,0,-10),v30,z10,DrillTool\WObj:=FakeWing;
        MoveL RelTool(Target_2310,0,0,-10),v30,z10,DrillTool\WObj:=FakeWing;
        MoveL Target_2310,v30,fine,DrillTool\WObj:=FakeWing;
SetDO drillDone,1;
WaitUntil drillDone = 0;
        MoveL RelTool(Target_2310,0,0,-10),v30,z10,DrillTool\WObj:=FakeWing;
        MoveL RelTool(Target_2320,0,0,-10),v30,z10,DrillTool\WObj:=FakeWing;
        MoveL Target_2320,v30,fine,DrillTool\WObj:=FakeWing;
SetDO drillDone,1;
WaitUntil drillDone = 0;
        MoveL RelTool(Target_2320,0,0,-10),v30,z10,DrillTool\WObj:=FakeWing;
        MoveL RelTool(Target_2330,0,0,-10),v30,z10,DrillTool\WObj:=FakeWing;
        MoveL Target_2330,v30,fine,DrillTool\WObj:=FakeWing;
SetDO drillDone,1;
WaitUntil drillDone = 0;
        MoveL RelTool(Target_2330,0,0,-10),v30,z10,DrillTool\WObj:=FakeWing;
        MoveL RelTool(Target_2340,0,0,-10),v30,z10,DrillTool\WObj:=FakeWing;
        MoveL Target_2340,v30,fine,DrillTool\WObj:=FakeWing;
SetDO drillDone,1;
WaitUntil drillDone = 0;
        MoveL RelTool(Target_2340,0,0,-10),v30,z10,DrillTool\WObj:=FakeWing;
        MoveL RelTool(Target_2350,0,0,-10),v30,z10,DrillTool\WObj:=FakeWing;
        MoveL Target_2350,v30,fine,DrillTool\WObj:=FakeWing;
SetDO drillDone,1;
WaitUntil drillDone = 0;
        MoveL RelTool(Target_2350,0,0,-10),v30,z10,DrillTool\WObj:=FakeWing;
        MoveL RelTool(Target_2360,0,0,-10),v30,z10,DrillTool\WObj:=FakeWing;
        MoveL Target_2360,v30,fine,DrillTool\WObj:=FakeWing;
SetDO drillDone,1;
WaitUntil drillDone = 0;
        MoveL RelTool(Target_2360,0,0,-10),v30,z10,DrillTool\WObj:=FakeWing;
        MoveL RelTool(Target_2370,0,0,-10),v30,z10,DrillTool\WObj:=FakeWing;
        MoveL Target_2370,v30,fine,DrillTool\WObj:=FakeWing;
SetDO drillDone,1;
WaitUntil drillDone = 0;
        MoveL RelTool(Target_2370,0,0,-10),v30,z10,DrillTool\WObj:=FakeWing;
        MoveL RelTool(Target_2380,0,0,-10),v30,z10,DrillTool\WObj:=FakeWing;
        MoveL Target_2380,v30,fine,DrillTool\WObj:=FakeWing;
SetDO drillDone,1;
WaitUntil drillDone = 0;
        MoveL RelTool(Target_2380,0,0,-10),v30,z10,DrillTool\WObj:=FakeWing;
        MoveL RelTool(Target_2390,0,0,-10),v30,z10,DrillTool\WObj:=FakeWing;
        MoveL Target_2390,v30,fine,DrillTool\WObj:=FakeWing;
SetDO drillDone,1;
WaitUntil drillDone = 0;
        MoveL RelTool(Target_2390,0,0,-10),v30,z10,DrillTool\WObj:=FakeWing;
        MoveL RelTool(Target_2400,0,0,-10),v30,z10,DrillTool\WObj:=FakeWing;
        MoveL Target_2400,v30,fine,DrillTool\WObj:=FakeWing;
SetDO drillDone,1;
WaitUntil drillDone = 0;
        MoveL RelTool(Target_2400,0,0,-10),v30,z10,DrillTool\WObj:=FakeWing;
        MoveL RelTool(Target_2410,0,0,-10),v30,z10,DrillTool\WObj:=FakeWing;
        MoveL Target_2410,v30,fine,DrillTool\WObj:=FakeWing;
SetDO drillDone,1;
WaitUntil drillDone = 0;
        MoveL RelTool(Target_2410,0,0,-10),v30,z10,DrillTool\WObj:=FakeWing;
        MoveL RelTool(Target_2420,0,0,-10),v30,z10,DrillTool\WObj:=FakeWing;
        MoveL Target_2420,v30,fine,DrillTool\WObj:=FakeWing;
SetDO drillDone,1;
WaitUntil drillDone = 0;
        MoveL RelTool(Target_2420,0,0,-10),v30,z10,DrillTool\WObj:=FakeWing;
        MoveL RelTool(Target_2430,0,0,-10),v30,z10,DrillTool\WObj:=FakeWing;
        MoveL Target_2430,v30,fine,DrillTool\WObj:=FakeWing;
SetDO drillDone,1;
WaitUntil drillDone = 0;
        MoveL RelTool(Target_2430,0,0,-10),v30,z10,DrillTool\WObj:=FakeWing;
        MoveL RelTool(Target_2440,0,0,-10),v30,z10,DrillTool\WObj:=FakeWing;
        MoveL Target_2440,v30,fine,DrillTool\WObj:=FakeWing;
SetDO drillDone,1;
WaitUntil drillDone = 0;
        MoveL RelTool(Target_2440,0,0,-10),v30,z10,DrillTool\WObj:=FakeWing;
        MoveL RelTool(Target_2450,0,0,-10),v30,z10,DrillTool\WObj:=FakeWing;
        MoveL Target_2450,v30,fine,DrillTool\WObj:=FakeWing;
SetDO drillDone,1;
WaitUntil drillDone = 0;
        MoveL RelTool(Target_2450,0,0,-10),v30,z10,DrillTool\WObj:=FakeWing;
        MoveL RelTool(Target_2460,0,0,-10),v30,z10,DrillTool\WObj:=FakeWing;
        MoveL Target_2460,v30,fine,DrillTool\WObj:=FakeWing;
SetDO drillDone,1;
WaitUntil drillDone = 0;
        MoveL RelTool(Target_2460,0,0,-10),v30,z10,DrillTool\WObj:=FakeWing;
        MoveL RelTool(Target_2470,0,0,-10),v30,z10,DrillTool\WObj:=FakeWing;
        MoveL Target_2470,v30,fine,DrillTool\WObj:=FakeWing;
SetDO drillDone,1;
WaitUntil drillDone = 0;
        MoveL RelTool(Target_2470,0,0,-10),v30,z10,DrillTool\WObj:=FakeWing;
        MoveL RelTool(Target_2480,0,0,-10),v30,z10,DrillTool\WObj:=FakeWing;
        MoveL Target_2480,v30,fine,DrillTool\WObj:=FakeWing;
SetDO drillDone,1;
WaitUntil drillDone = 0;
        MoveL RelTool(Target_2480,0,0,-10),v30,z10,DrillTool\WObj:=FakeWing;
        MoveL RelTool(Target_2490,0,0,-10),v30,z10,DrillTool\WObj:=FakeWing;
        MoveL Target_2490,v30,fine,DrillTool\WObj:=FakeWing;
SetDO drillDone,1;
WaitUntil drillDone = 0;
        MoveL RelTool(Target_2490,0,0,-10),v30,z10,DrillTool\WObj:=FakeWing;
        MoveL RelTool(Target_2500,0,0,-10),v30,z10,DrillTool\WObj:=FakeWing;
        MoveL Target_2500,v30,fine,DrillTool\WObj:=FakeWing;
SetDO drillDone,1;
WaitUntil drillDone = 0;
        MoveL RelTool(Target_2500,0,0,-10),v30,z10,DrillTool\WObj:=FakeWing;
        MoveL RelTool(Target_2510,0,0,-10),v30,z10,DrillTool\WObj:=FakeWing;
        MoveL Target_2510,v30,fine,DrillTool\WObj:=FakeWing;
SetDO drillDone,1;
WaitUntil drillDone = 0;
        MoveL RelTool(Target_2510,0,0,-10),v30,z10,DrillTool\WObj:=FakeWing;
        MoveL RelTool(Target_2520,0,0,-10),v30,z10,DrillTool\WObj:=FakeWing;
        MoveL Target_2520,v30,fine,DrillTool\WObj:=FakeWing;
SetDO drillDone,1;
WaitUntil drillDone = 0;
        MoveL RelTool(Target_2520,0,0,-10),v30,z10,DrillTool\WObj:=FakeWing;
        MoveL RelTool(Target_2530,0,0,-10),v30,z10,DrillTool\WObj:=FakeWing;
        MoveL Target_2530,v30,fine,DrillTool\WObj:=FakeWing;
SetDO drillDone,1;
WaitUntil drillDone = 0;
        MoveL RelTool(Target_2530,0,0,-10),v30,z10,DrillTool\WObj:=FakeWing;
        MoveL RelTool(Target_2540,0,0,-10),v30,z10,DrillTool\WObj:=FakeWing;
        MoveL Target_2540,v30,fine,DrillTool\WObj:=FakeWing;
SetDO drillDone,1;
WaitUntil drillDone = 0;
        MoveL RelTool(Target_2540,0,0,-10),v30,z10,DrillTool\WObj:=FakeWing;
        MoveL RelTool(Target_2550,0,0,-10),v30,z10,DrillTool\WObj:=FakeWing;
        MoveL Target_2550,v30,fine,DrillTool\WObj:=FakeWing;
SetDO drillDone,1;
WaitUntil drillDone = 0;
        MoveL RelTool(Target_2550,0,0,-10),v30,z10,DrillTool\WObj:=FakeWing;
        MoveL RelTool(Target_2560,0,0,-10),v30,z10,DrillTool\WObj:=FakeWing;
        MoveL Target_2560,v30,fine,DrillTool\WObj:=FakeWing;
SetDO drillDone,1;
WaitUntil drillDone = 0;
        MoveL RelTool(Target_2560,0,0,-10),v30,z10,DrillTool\WObj:=FakeWing;
        MoveL RelTool(Target_2570,0,0,-10),v30,z10,DrillTool\WObj:=FakeWing;
        MoveL Target_2570,v30,fine,DrillTool\WObj:=FakeWing;
SetDO drillDone,1;
WaitUntil drillDone = 0;
        MoveL RelTool(Target_2570,0,0,-10),v30,z10,DrillTool\WObj:=FakeWing;
        MoveL RelTool(Target_2580,0,0,-10),v30,z10,DrillTool\WObj:=FakeWing;
        MoveL Target_2580,v30,fine,DrillTool\WObj:=FakeWing;
SetDO drillDone,1;
WaitUntil drillDone = 0;
        MoveL RelTool(Target_2580,0,0,-10),v30,z10,DrillTool\WObj:=FakeWing;
        MoveL RelTool(Target_2590,0,0,-10),v30,z10,DrillTool\WObj:=FakeWing;
        MoveL Target_2590,v30,fine,DrillTool\WObj:=FakeWing;
SetDO drillDone,1;
WaitUntil drillDone = 0;
        MoveL RelTool(Target_2590,0,0,-10),v30,z10,DrillTool\WObj:=FakeWing;
        MoveL RelTool(Target_2600,0,0,-10),v30,z10,DrillTool\WObj:=FakeWing;
        MoveL Target_2600,v30,fine,DrillTool\WObj:=FakeWing;
SetDO drillDone,1;
WaitUntil drillDone = 0;
        MoveL RelTool(Target_2600,0,0,-10),v30,z10,DrillTool\WObj:=FakeWing;
        MoveL RelTool(Target_2610,0,0,-10),v30,z10,DrillTool\WObj:=FakeWing;
        MoveL Target_2610,v30,fine,DrillTool\WObj:=FakeWing;
SetDO drillDone,1;
WaitUntil drillDone = 0;
        MoveL RelTool(Target_2610,0,0,-10),v30,z10,DrillTool\WObj:=FakeWing;
        MoveL RelTool(Target_2620,0,0,-10),v30,z10,DrillTool\WObj:=FakeWing;
        MoveL Target_2620,v30,fine,DrillTool\WObj:=FakeWing;
SetDO drillDone,1;
WaitUntil drillDone = 0;
        MoveL RelTool(Target_2620,0,0,-10),v30,z10,DrillTool\WObj:=FakeWing;
        MoveL RelTool(Target_2630,0,0,-10),v30,z10,DrillTool\WObj:=FakeWing;
        MoveL Target_2630,v30,fine,DrillTool\WObj:=FakeWing;
SetDO drillDone,1;
WaitUntil drillDone = 0;
        MoveL RelTool(Target_2630,0,0,-10),v30,z10,DrillTool\WObj:=FakeWing;
        MoveL RelTool(Target_2640,0,0,-10),v30,z10,DrillTool\WObj:=FakeWing;
        MoveL Target_2640,v30,fine,DrillTool\WObj:=FakeWing;
SetDO drillDone,1;
WaitUntil drillDone = 0;
        MoveL RelTool(Target_2640,0,0,-10),v30,z10,DrillTool\WObj:=FakeWing;
        MoveL RelTool(Target_2650,0,0,-10),v30,z10,DrillTool\WObj:=FakeWing;
        MoveL Target_2650,v30,fine,DrillTool\WObj:=FakeWing;
SetDO drillDone,1;
WaitUntil drillDone = 0;
        MoveL RelTool(Target_2650,0,0,-10),v30,z10,DrillTool\WObj:=FakeWing;
        MoveL RelTool(Target_2660,0,0,-10),v30,z10,DrillTool\WObj:=FakeWing;
        MoveL Target_2660,v30,fine,DrillTool\WObj:=FakeWing;
SetDO drillDone,1;
WaitUntil drillDone = 0;
        MoveL RelTool(Target_2660,0,0,-10),v30,z10,DrillTool\WObj:=FakeWing;
        MoveL RelTool(Target_2670,0,0,-10),v30,z10,DrillTool\WObj:=FakeWing;
        MoveL Target_2670,v30,fine,DrillTool\WObj:=FakeWing;
SetDO drillDone,1;
WaitUntil drillDone = 0;
        MoveL RelTool(Target_2670,0,0,-10),v30,z10,DrillTool\WObj:=FakeWing;
        MoveL RelTool(Target_2680,0,0,-10),v30,z10,DrillTool\WObj:=FakeWing;
        MoveL Target_2680,v30,fine,DrillTool\WObj:=FakeWing;
SetDO drillDone,1;
WaitUntil drillDone = 0;
        MoveL RelTool(Target_2680,0,0,-10),v30,z10,DrillTool\WObj:=FakeWing;
        MoveL RelTool(Target_2690,0,0,-10),v30,z10,DrillTool\WObj:=FakeWing;
        MoveL Target_2690,v30,fine,DrillTool\WObj:=FakeWing;
SetDO drillDone,1;
WaitUntil drillDone = 0;
        MoveL RelTool(Target_2690,0,0,-10),v30,z10,DrillTool\WObj:=FakeWing;
        MoveL RelTool(Target_2700,0,0,-10),v30,z10,DrillTool\WObj:=FakeWing;
        MoveL Target_2700,v30,fine,DrillTool\WObj:=FakeWing;
SetDO drillDone,1;
WaitUntil drillDone = 0;
        MoveL RelTool(Target_2700,0,0,-10),v30,z10,DrillTool\WObj:=FakeWing;
        MoveL RelTool(Target_2710,0,0,-10),v30,z10,DrillTool\WObj:=FakeWing;
        MoveL Target_2710,v30,fine,DrillTool\WObj:=FakeWing;
SetDO drillDone,1;
WaitUntil drillDone = 0;
        MoveL RelTool(Target_2710,0,0,-10),v30,z10,DrillTool\WObj:=FakeWing;
        MoveL RelTool(Target_2720,0,0,-10),v30,z10,DrillTool\WObj:=FakeWing;
        MoveL Target_2720,v30,fine,DrillTool\WObj:=FakeWing;
SetDO drillDone,1;
WaitUntil drillDone = 0;
        MoveL RelTool(Target_2720,0,0,-10),v30,z10,DrillTool\WObj:=FakeWing;
        MoveL RelTool(Target_2730,0,0,-10),v30,z10,DrillTool\WObj:=FakeWing;
        MoveL Target_2730,v30,fine,DrillTool\WObj:=FakeWing;
SetDO drillDone,1;
WaitUntil drillDone = 0;
        MoveL RelTool(Target_2730,0,0,-10),v30,z10,DrillTool\WObj:=FakeWing;
        MoveL RelTool(Target_2740,0,0,-10),v30,z10,DrillTool\WObj:=FakeWing;
        MoveL Target_2740,v30,fine,DrillTool\WObj:=FakeWing;
SetDO drillDone,1;
WaitUntil drillDone = 0;
        MoveL RelTool(Target_2740,0,0,-10),v30,z10,DrillTool\WObj:=FakeWing;
        MoveL RelTool(Target_2750,0,0,-10),v30,z10,DrillTool\WObj:=FakeWing;
        MoveL Target_2750,v30,fine,DrillTool\WObj:=FakeWing;
SetDO drillDone,1;
WaitUntil drillDone = 0;
        MoveL RelTool(Target_2750,0,0,-10),v30,z10,DrillTool\WObj:=FakeWing;
        MoveL RelTool(Target_2760,0,0,-10),v30,z10,DrillTool\WObj:=FakeWing;
        MoveL Target_2760,v30,fine,DrillTool\WObj:=FakeWing;
SetDO drillDone,1;
WaitUntil drillDone = 0;
        MoveL RelTool(Target_2760,0,0,-10),v30,z10,DrillTool\WObj:=FakeWing;
        MoveL RelTool(Target_2770,0,0,-10),v30,z10,DrillTool\WObj:=FakeWing;
        MoveL Target_2770,v30,fine,DrillTool\WObj:=FakeWing;
SetDO drillDone,1;
WaitUntil drillDone = 0;
        MoveL RelTool(Target_2770,0,0,-10),v30,z10,DrillTool\WObj:=FakeWing;
        MoveL RelTool(Target_2780,0,0,-10),v30,z10,DrillTool\WObj:=FakeWing;
        MoveL Target_2780,v30,fine,DrillTool\WObj:=FakeWing;
SetDO drillDone,1;
WaitUntil drillDone = 0;
        MoveL RelTool(Target_2780,0,0,-10),v30,z10,DrillTool\WObj:=FakeWing;
        MoveL RelTool(Target_2790,0,0,-10),v30,z10,DrillTool\WObj:=FakeWing;
        MoveL Target_2790,v30,fine,DrillTool\WObj:=FakeWing;
SetDO drillDone,1;
WaitUntil drillDone = 0;
        MoveL RelTool(Target_2790,0,0,-10),v30,z10,DrillTool\WObj:=FakeWing;
        MoveL RelTool(Target_2800,0,0,-10),v30,z10,DrillTool\WObj:=FakeWing;
        MoveL Target_2800,v30,fine,DrillTool\WObj:=FakeWing;
SetDO drillDone,1;
WaitUntil drillDone = 0;
        MoveL RelTool(Target_2800,0,0,-10),v30,z10,DrillTool\WObj:=FakeWing;
        MoveL RelTool(Target_2810,0,0,-10),v30,z10,DrillTool\WObj:=FakeWing;
        MoveL Target_2810,v30,fine,DrillTool\WObj:=FakeWing;
SetDO drillDone,1;
WaitUntil drillDone = 0;
        MoveL RelTool(Target_2810,0,0,-10),v30,z10,DrillTool\WObj:=FakeWing;
        MoveL RelTool(Target_2820,0,0,-10),v30,z10,DrillTool\WObj:=FakeWing;
        MoveL Target_2820,v30,fine,DrillTool\WObj:=FakeWing;
SetDO drillDone,1;
WaitUntil drillDone = 0;
        MoveL RelTool(Target_2820,0,0,-10),v30,z10,DrillTool\WObj:=FakeWing;
        MoveL RelTool(Target_2830,0,0,-10),v30,z10,DrillTool\WObj:=FakeWing;
        MoveL Target_2830,v30,fine,DrillTool\WObj:=FakeWing;
SetDO drillDone,1;
WaitUntil drillDone = 0;
        MoveL RelTool(Target_2830,0,0,-10),v30,z10,DrillTool\WObj:=FakeWing;
        MoveL RelTool(Target_2840,0,0,-10),v30,z10,DrillTool\WObj:=FakeWing;
        MoveL Target_2840,v30,fine,DrillTool\WObj:=FakeWing;
SetDO drillDone,1;
WaitUntil drillDone = 0;
        MoveL RelTool(Target_2840,0,0,-10),v30,z10,DrillTool\WObj:=FakeWing;
        MoveL RelTool(Target_2850,0,0,-10),v30,z10,DrillTool\WObj:=FakeWing;
        MoveL Target_2850,v30,fine,DrillTool\WObj:=FakeWing;
SetDO drillDone,1;
WaitUntil drillDone = 0;
        MoveL RelTool(Target_2850,0,0,-10),v30,z10,DrillTool\WObj:=FakeWing;
        MoveL RelTool(Target_2860,0,0,-10),v30,z10,DrillTool\WObj:=FakeWing;
        MoveL Target_2860,v30,fine,DrillTool\WObj:=FakeWing;
SetDO drillDone,1;
WaitUntil drillDone = 0;
        MoveL RelTool(Target_2860,0,0,-10),v30,z10,DrillTool\WObj:=FakeWing;
        MoveL RelTool(Target_2870,0,0,-10),v30,z10,DrillTool\WObj:=FakeWing;
        MoveL Target_2870,v30,fine,DrillTool\WObj:=FakeWing;
SetDO drillDone,1;
WaitUntil drillDone = 0;
        MoveL RelTool(Target_2870,0,0,-10),v30,z10,DrillTool\WObj:=FakeWing;
        MoveL RelTool(Target_2880,0,0,-10),v30,z10,DrillTool\WObj:=FakeWing;
        MoveL Target_2880,v30,fine,DrillTool\WObj:=FakeWing;
SetDO drillDone,1;
WaitUntil drillDone = 0;
        MoveL RelTool(Target_2880,0,0,-10),v30,z10,DrillTool\WObj:=FakeWing;
        MoveL RelTool(Target_2890,0,0,-10),v30,z10,DrillTool\WObj:=FakeWing;
        MoveL Target_2890,v30,fine,DrillTool\WObj:=FakeWing;
SetDO drillDone,1;
WaitUntil drillDone = 0;
        MoveL RelTool(Target_2890,0,0,-10),v30,z10,DrillTool\WObj:=FakeWing;
        MoveL RelTool(Target_2900,0,0,-10),v30,z10,DrillTool\WObj:=FakeWing;
        MoveL Target_2900,v30,fine,DrillTool\WObj:=FakeWing;
SetDO drillDone,1;
WaitUntil drillDone = 0;
        MoveL RelTool(Target_2900,0,0,-10),v30,z10,DrillTool\WObj:=FakeWing;
        MoveL RelTool(Target_2910,0,0,-10),v30,z10,DrillTool\WObj:=FakeWing;
        MoveL Target_2910,v30,fine,DrillTool\WObj:=FakeWing;
SetDO drillDone,1;
WaitUntil drillDone = 0;
        MoveL RelTool(Target_2910,0,0,-10),v30,z10,DrillTool\WObj:=FakeWing;
        MoveL RelTool(Target_2920,0,0,-10),v30,z10,DrillTool\WObj:=FakeWing;
        MoveL Target_2920,v30,fine,DrillTool\WObj:=FakeWing;
SetDO drillDone,1;
WaitUntil drillDone = 0;
        MoveL RelTool(Target_2920,0,0,-10),v30,z10,DrillTool\WObj:=FakeWing;
        MoveL RelTool(Target_2930,0,0,-10),v30,z10,DrillTool\WObj:=FakeWing;
        MoveL Target_2930,v30,fine,DrillTool\WObj:=FakeWing;
SetDO drillDone,1;
WaitUntil drillDone = 0;
        MoveL RelTool(Target_2930,0,0,-10),v30,z10,DrillTool\WObj:=FakeWing;
        MoveL RelTool(Target_2940,0,0,-10),v30,z10,DrillTool\WObj:=FakeWing;
        MoveL Target_2940,v30,fine,DrillTool\WObj:=FakeWing;
SetDO drillDone,1;
WaitUntil drillDone = 0;
        MoveL RelTool(Target_2940,0,0,-10),v30,z10,DrillTool\WObj:=FakeWing;
        MoveL RelTool(Target_2950,0,0,-10),v30,z10,DrillTool\WObj:=FakeWing;
        MoveL Target_2950,v30,fine,DrillTool\WObj:=FakeWing;
SetDO drillDone,1;
WaitUntil drillDone = 0;
        MoveL RelTool(Target_2950,0,0,-10),v30,z10,DrillTool\WObj:=FakeWing;
        MoveL RelTool(Target_2960,0,0,-10),v30,z10,DrillTool\WObj:=FakeWing;
        MoveL Target_2960,v30,fine,DrillTool\WObj:=FakeWing;
SetDO drillDone,1;
WaitUntil drillDone = 0;
        MoveL RelTool(Target_2960,0,0,-10),v30,z10,DrillTool\WObj:=FakeWing;
        MoveL RelTool(Target_2970,0,0,-10),v30,z10,DrillTool\WObj:=FakeWing;
        MoveL Target_2970,v30,fine,DrillTool\WObj:=FakeWing;
SetDO drillDone,1;
WaitUntil drillDone = 0;
        MoveL RelTool(Target_2970,0,0,-10),v30,z10,DrillTool\WObj:=FakeWing;
        MoveL RelTool(Target_2980,0,0,-10),v30,z10,DrillTool\WObj:=FakeWing;
        MoveL Target_2980,v30,fine,DrillTool\WObj:=FakeWing;
SetDO drillDone,1;
WaitUntil drillDone = 0;
        MoveL RelTool(Target_2980,0,0,-10),v30,z10,DrillTool\WObj:=FakeWing;
        MoveL RelTool(Target_2990,0,0,-10),v30,z10,DrillTool\WObj:=FakeWing;
        MoveL Target_2990,v30,fine,DrillTool\WObj:=FakeWing;
SetDO drillDone,1;
WaitUntil drillDone = 0;
        MoveL RelTool(Target_2990,0,0,-10),v30,z10,DrillTool\WObj:=FakeWing;
        MoveL RelTool(Target_3000,0,0,-10),v30,z10,DrillTool\WObj:=FakeWing;
        MoveL Target_3000,v30,fine,DrillTool\WObj:=FakeWing;
SetDO drillDone,1;
WaitUntil drillDone = 0;
        MoveL RelTool(Target_3000,0,0,-10),v30,z10,DrillTool\WObj:=FakeWing;
        MoveL RelTool(Target_3010,0,0,-10),v30,z10,DrillTool\WObj:=FakeWing;
        MoveL Target_3010,v30,fine,DrillTool\WObj:=FakeWing;
SetDO drillDone,1;
WaitUntil drillDone = 0;
        MoveL RelTool(Target_3010,0,0,-10),v30,z10,DrillTool\WObj:=FakeWing;
        MoveL RelTool(Target_3020,0,0,-10),v30,z10,DrillTool\WObj:=FakeWing;
        MoveL Target_3020,v30,fine,DrillTool\WObj:=FakeWing;
SetDO drillDone,1;
WaitUntil drillDone = 0;
        MoveL RelTool(Target_3020,0,0,-10),v30,z10,DrillTool\WObj:=FakeWing;
        MoveL RelTool(Target_3030,0,0,-10),v30,z10,DrillTool\WObj:=FakeWing;
        MoveL Target_3030,v30,fine,DrillTool\WObj:=FakeWing;
SetDO drillDone,1;
WaitUntil drillDone = 0;
        MoveL RelTool(Target_3030,0,0,-10),v30,z10,DrillTool\WObj:=FakeWing;
        MoveL RelTool(Target_3040,0,0,-10),v30,z10,DrillTool\WObj:=FakeWing;
        MoveL Target_3040,v30,fine,DrillTool\WObj:=FakeWing;
SetDO drillDone,1;
WaitUntil drillDone = 0;
        MoveL RelTool(Target_3040,0,0,-10),v30,z10,DrillTool\WObj:=FakeWing;
        MoveL RelTool(Target_3050,0,0,-10),v30,z10,DrillTool\WObj:=FakeWing;
        MoveL Target_3050,v30,fine,DrillTool\WObj:=FakeWing;
SetDO drillDone,1;
WaitUntil drillDone = 0;
        MoveL RelTool(Target_3050,0,0,-10),v30,z10,DrillTool\WObj:=FakeWing;
        MoveL RelTool(Target_3060,0,0,-10),v30,z10,DrillTool\WObj:=FakeWing;
        MoveL Target_3060,v30,fine,DrillTool\WObj:=FakeWing;
SetDO drillDone,1;
WaitUntil drillDone = 0;
        MoveL RelTool(Target_3060,0,0,-10),v30,z10,DrillTool\WObj:=FakeWing;
        MoveL RelTool(Target_3070,0,0,-10),v30,z10,DrillTool\WObj:=FakeWing;
        MoveL Target_3070,v30,fine,DrillTool\WObj:=FakeWing;
SetDO drillDone,1;
WaitUntil drillDone = 0;
        MoveL RelTool(Target_3070,0,0,-10),v30,z10,DrillTool\WObj:=FakeWing;
        MoveL RelTool(Target_3080,0,0,-10),v30,z10,DrillTool\WObj:=FakeWing;
        MoveL Target_3080,v30,fine,DrillTool\WObj:=FakeWing;
SetDO drillDone,1;
WaitUntil drillDone = 0;
        MoveL RelTool(Target_3080,0,0,-10),v30,z10,DrillTool\WObj:=FakeWing;
        MoveL RelTool(Target_3090,0,0,-10),v30,z10,DrillTool\WObj:=FakeWing;
        MoveL Target_3090,v30,fine,DrillTool\WObj:=FakeWing;
SetDO drillDone,1;
WaitUntil drillDone = 0;
        MoveL RelTool(Target_3090,0,0,-10),v30,z10,DrillTool\WObj:=FakeWing;
        MoveL RelTool(Target_3100,0,0,-10),v30,z10,DrillTool\WObj:=FakeWing;
        MoveL Target_3100,v30,fine,DrillTool\WObj:=FakeWing;
SetDO drillDone,1;
WaitUntil drillDone = 0;
        MoveL RelTool(Target_3100,0,0,-10),v30,z10,DrillTool\WObj:=FakeWing;
        MoveL RelTool(Target_3110,0,0,-10),v30,z10,DrillTool\WObj:=FakeWing;
        MoveL Target_3110,v30,fine,DrillTool\WObj:=FakeWing;
SetDO drillDone,1;
WaitUntil drillDone = 0;
        MoveL RelTool(Target_3110,0,0,-10),v30,z10,DrillTool\WObj:=FakeWing;
        MoveL RelTool(Target_3120,0,0,-10),v30,z10,DrillTool\WObj:=FakeWing;
        MoveL Target_3120,v30,fine,DrillTool\WObj:=FakeWing;
SetDO drillDone,1;
WaitUntil drillDone = 0;
        MoveL RelTool(Target_3120,0,0,-10),v30,z10,DrillTool\WObj:=FakeWing;
        MoveL RelTool(Target_3130,0,0,-10),v30,z10,DrillTool\WObj:=FakeWing;
        MoveL Target_3130,v30,fine,DrillTool\WObj:=FakeWing;
SetDO drillDone,1;
WaitUntil drillDone = 0;
        MoveL RelTool(Target_3130,0,0,-10),v30,z10,DrillTool\WObj:=FakeWing;
        MoveL RelTool(Target_3140,0,0,-10),v30,z10,DrillTool\WObj:=FakeWing;
        MoveL Target_3140,v30,fine,DrillTool\WObj:=FakeWing;
SetDO drillDone,1;
WaitUntil drillDone = 0;
        MoveL RelTool(Target_3140,0,0,-10),v30,z10,DrillTool\WObj:=FakeWing;
        MoveL RelTool(Target_3150,0,0,-10),v30,z10,DrillTool\WObj:=FakeWing;
        MoveL Target_3150,v30,fine,DrillTool\WObj:=FakeWing;
SetDO drillDone,1;
WaitUntil drillDone = 0;
        MoveL RelTool(Target_3150,0,0,-10),v30,z10,DrillTool\WObj:=FakeWing;
        MoveL RelTool(Target_3160,0,0,-10),v30,z10,DrillTool\WObj:=FakeWing;
        MoveL Target_3160,v30,fine,DrillTool\WObj:=FakeWing;
SetDO drillDone,1;
WaitUntil drillDone = 0;
        MoveL RelTool(Target_3160,0,0,-10),v30,z10,DrillTool\WObj:=FakeWing;
        MoveL RelTool(Target_3170,0,0,-10),v30,z10,DrillTool\WObj:=FakeWing;
        MoveL Target_3170,v30,fine,DrillTool\WObj:=FakeWing;
SetDO drillDone,1;
WaitUntil drillDone = 0;
        MoveL RelTool(Target_3170,0,0,-10),v30,z10,DrillTool\WObj:=FakeWing;
        MoveL RelTool(Target_3180,0,0,-10),v30,z10,DrillTool\WObj:=FakeWing;
        MoveL Target_3180,v30,fine,DrillTool\WObj:=FakeWing;
SetDO drillDone,1;
WaitUntil drillDone = 0;
        MoveL RelTool(Target_3180,0,0,-10),v30,z10,DrillTool\WObj:=FakeWing;
        MoveL RelTool(Target_3190,0,0,-10),v30,z10,DrillTool\WObj:=FakeWing;
        MoveL Target_3190,v30,fine,DrillTool\WObj:=FakeWing;
SetDO drillDone,1;
WaitUntil drillDone = 0;
        MoveL RelTool(Target_3190,0,0,-10),v30,z10,DrillTool\WObj:=FakeWing;
        MoveL RelTool(Target_3200,0,0,-10),v30,z10,DrillTool\WObj:=FakeWing;
        MoveL Target_3200,v30,fine,DrillTool\WObj:=FakeWing;
SetDO drillDone,1;
WaitUntil drillDone = 0;
        MoveL RelTool(Target_3200,0,0,-10),v30,z10,DrillTool\WObj:=FakeWing;
        MoveL RelTool(Target_3210,0,0,-10),v30,z10,DrillTool\WObj:=FakeWing;
        MoveL Target_3210,v30,fine,DrillTool\WObj:=FakeWing;
SetDO drillDone,1;
WaitUntil drillDone = 0;
        MoveL RelTool(Target_3210,0,0,-10),v30,z10,DrillTool\WObj:=FakeWing;
        MoveL RelTool(Target_3220,0,0,-10),v30,z10,DrillTool\WObj:=FakeWing;
        MoveL Target_3220,v30,fine,DrillTool\WObj:=FakeWing;
SetDO drillDone,1;
WaitUntil drillDone = 0;
        MoveL RelTool(Target_3220,0,0,-10),v30,z10,DrillTool\WObj:=FakeWing;
        MoveL RelTool(Target_3230,0,0,-10),v30,z10,DrillTool\WObj:=FakeWing;
        MoveL Target_3230,v30,fine,DrillTool\WObj:=FakeWing;
SetDO drillDone,1;
WaitUntil drillDone = 0;
        MoveL RelTool(Target_3230,0,0,-10),v30,z10,DrillTool\WObj:=FakeWing;
        MoveL RelTool(Target_3240,0,0,-10),v30,z10,DrillTool\WObj:=FakeWing;
        MoveL Target_3240,v30,fine,DrillTool\WObj:=FakeWing;
SetDO drillDone,1;
WaitUntil drillDone = 0;
        MoveL RelTool(Target_3240,0,0,-10),v30,z10,DrillTool\WObj:=FakeWing;
        MoveL RelTool(Target_3250,0,0,-10),v30,z10,DrillTool\WObj:=FakeWing;
        MoveL Target_3250,v30,fine,DrillTool\WObj:=FakeWing;
SetDO drillDone,1;
WaitUntil drillDone = 0;
        MoveL RelTool(Target_3250,0,0,-10),v30,z10,DrillTool\WObj:=FakeWing;
        MoveL RelTool(Target_3260,0,0,-10),v30,z10,DrillTool\WObj:=FakeWing;
        MoveL Target_3260,v30,fine,DrillTool\WObj:=FakeWing;
SetDO drillDone,1;
WaitUntil drillDone = 0;
        MoveL RelTool(Target_3260,0,0,-10),v30,z10,DrillTool\WObj:=FakeWing;
        MoveL RelTool(Target_3270,0,0,-10),v30,z10,DrillTool\WObj:=FakeWing;
        MoveL Target_3270,v30,fine,DrillTool\WObj:=FakeWing;
SetDO drillDone,1;
WaitUntil drillDone = 0;
        MoveL RelTool(Target_3270,0,0,-10),v30,z10,DrillTool\WObj:=FakeWing;
        MoveL RelTool(Target_3280,0,0,-10),v30,z10,DrillTool\WObj:=FakeWing;
        MoveL Target_3280,v30,fine,DrillTool\WObj:=FakeWing;
SetDO drillDone,1;
WaitUntil drillDone = 0;
        MoveL RelTool(Target_3280,0,0,-10),v30,z10,DrillTool\WObj:=FakeWing;
        MoveL RelTool(Target_3290,0,0,-10),v30,z10,DrillTool\WObj:=FakeWing;
        MoveL Target_3290,v30,fine,DrillTool\WObj:=FakeWing;
SetDO drillDone,1;
WaitUntil drillDone = 0;
        MoveL RelTool(Target_3290,0,0,-10),v30,z10,DrillTool\WObj:=FakeWing;
        MoveL RelTool(Target_3300,0,0,-10),v30,z10,DrillTool\WObj:=FakeWing;
        MoveL Target_3300,v30,fine,DrillTool\WObj:=FakeWing;
SetDO drillDone,1;
WaitUntil drillDone = 0;
        MoveL RelTool(Target_3300,0,0,-10),v30,z10,DrillTool\WObj:=FakeWing;
        MoveL RelTool(Target_3310,0,0,-10),v30,z10,DrillTool\WObj:=FakeWing;
        MoveL Target_3310,v30,fine,DrillTool\WObj:=FakeWing;
SetDO drillDone,1;
WaitUntil drillDone = 0;
        MoveL RelTool(Target_3310,0,0,-10),v30,z10,DrillTool\WObj:=FakeWing;
        MoveL RelTool(Target_3320,0,0,-10),v30,z10,DrillTool\WObj:=FakeWing;
        MoveL Target_3320,v30,fine,DrillTool\WObj:=FakeWing;
SetDO drillDone,1;
WaitUntil drillDone = 0;
        MoveL RelTool(Target_3320,0,0,-10),v30,z10,DrillTool\WObj:=FakeWing;
        MoveL RelTool(Target_3330,0,0,-10),v30,z10,DrillTool\WObj:=FakeWing;
        MoveL Target_3330,v30,fine,DrillTool\WObj:=FakeWing;
SetDO drillDone,1;
WaitUntil drillDone = 0;
        MoveL RelTool(Target_3330,0,0,-10),v30,z10,DrillTool\WObj:=FakeWing;
        MoveL RelTool(Target_3340,0,0,-10),v30,z10,DrillTool\WObj:=FakeWing;
        MoveL Target_3340,v30,fine,DrillTool\WObj:=FakeWing;
SetDO drillDone,1;
WaitUntil drillDone = 0;
        MoveL RelTool(Target_3340,0,0,-10),v30,z10,DrillTool\WObj:=FakeWing;
        MoveL RelTool(Target_3350,0,0,-10),v30,z10,DrillTool\WObj:=FakeWing;
        MoveL Target_3350,v30,fine,DrillTool\WObj:=FakeWing;
SetDO drillDone,1;
WaitUntil drillDone = 0;
        MoveL RelTool(Target_3350,0,0,-10),v30,z10,DrillTool\WObj:=FakeWing;
        MoveL RelTool(Target_3360,0,0,-10),v30,z10,DrillTool\WObj:=FakeWing;
        MoveL Target_3360,v30,fine,DrillTool\WObj:=FakeWing;
SetDO drillDone,1;
WaitUntil drillDone = 0;
        MoveL RelTool(Target_3360,0,0,-10),v30,z10,DrillTool\WObj:=FakeWing;
        MoveL RelTool(Target_3370,0,0,-10),v30,z10,DrillTool\WObj:=FakeWing;
        MoveL Target_3370,v30,fine,DrillTool\WObj:=FakeWing;
SetDO drillDone,1;
WaitUntil drillDone = 0;
        MoveL RelTool(Target_3370,0,0,-10),v30,z10,DrillTool\WObj:=FakeWing;
        MoveL RelTool(Target_3380,0,0,-10),v30,z10,DrillTool\WObj:=FakeWing;
        MoveL Target_3380,v30,fine,DrillTool\WObj:=FakeWing;
SetDO drillDone,1;
WaitUntil drillDone = 0;
        MoveL RelTool(Target_3380,0,0,-10),v30,z10,DrillTool\WObj:=FakeWing;
        MoveL RelTool(Target_3390,0,0,-10),v30,z10,DrillTool\WObj:=FakeWing;
        MoveL Target_3390,v30,fine,DrillTool\WObj:=FakeWing;
SetDO drillDone,1;
WaitUntil drillDone = 0;
        MoveL RelTool(Target_3390,0,0,-10),v30,z10,DrillTool\WObj:=FakeWing;
        MoveL RelTool(Target_3400,0,0,-10),v30,z10,DrillTool\WObj:=FakeWing;
        MoveL Target_3400,v30,fine,DrillTool\WObj:=FakeWing;
SetDO drillDone,1;
WaitUntil drillDone = 0;
        MoveL RelTool(Target_3400,0,0,-10),v30,z10,DrillTool\WObj:=FakeWing;
        MoveL RelTool(Target_3410,0,0,-10),v30,z10,DrillTool\WObj:=FakeWing;
        MoveL Target_3410,v30,fine,DrillTool\WObj:=FakeWing;
SetDO drillDone,1;
WaitUntil drillDone = 0;
        MoveL RelTool(Target_3410,0,0,-10),v30,z10,DrillTool\WObj:=FakeWing;
        MoveL RelTool(Target_3420,0,0,-10),v30,z10,DrillTool\WObj:=FakeWing;
        MoveL Target_3420,v30,fine,DrillTool\WObj:=FakeWing;
SetDO drillDone,1;
WaitUntil drillDone = 0;
        MoveL RelTool(Target_3420,0,0,-10),v30,z10,DrillTool\WObj:=FakeWing;
        MoveL RelTool(Target_3430,0,0,-10),v30,z10,DrillTool\WObj:=FakeWing;
        MoveL Target_3430,v30,fine,DrillTool\WObj:=FakeWing;
SetDO drillDone,1;
WaitUntil drillDone = 0;
        MoveL RelTool(Target_3430,0,0,-10),v30,z10,DrillTool\WObj:=FakeWing;
        MoveL RelTool(Target_3440,0,0,-10),v30,z10,DrillTool\WObj:=FakeWing;
        MoveL Target_3440,v30,fine,DrillTool\WObj:=FakeWing;
SetDO drillDone,1;
WaitUntil drillDone = 0;
        MoveL RelTool(Target_3440,0,0,-10),v30,z10,DrillTool\WObj:=FakeWing;
        MoveL RelTool(Target_3450,0,0,-10),v30,z10,DrillTool\WObj:=FakeWing;
        MoveL Target_3450,v30,fine,DrillTool\WObj:=FakeWing;
SetDO drillDone,1;
WaitUntil drillDone = 0;
        MoveL RelTool(Target_3450,0,0,-10),v30,z10,DrillTool\WObj:=FakeWing;
        MoveL RelTool(Target_3460,0,0,-10),v30,z10,DrillTool\WObj:=FakeWing;
        MoveL Target_3460,v30,fine,DrillTool\WObj:=FakeWing;
SetDO drillDone,1;
WaitUntil drillDone = 0;
        MoveL RelTool(Target_3460,0,0,-10),v30,z10,DrillTool\WObj:=FakeWing;
        MoveL RelTool(Target_3470,0,0,-10),v30,z10,DrillTool\WObj:=FakeWing;
        MoveL Target_3470,v30,fine,DrillTool\WObj:=FakeWing;
SetDO drillDone,1;
WaitUntil drillDone = 0;
